(* IEC 61131-3 sources: std_i2980_v2.06_cp053/Source/IMM/ieccontrol/ODC1 (part 5) *)

         IF bAllParallelOpenColumnsReady THEN
            fbDebugTrace2(nODCInterpreter, CONCAT('found fulfilled EndParallelOpen in column ',
                                                 DINT_TO_STRING(i),' -> increase row'));
            bIncreaseRow := TRUE;
         END_IF;

      ELSIF (MoveId  = cMoveNone) AND (MoveDir = cMoveNone) AND (DeviceId.CompId = cCompNone) THEN
         bIncreaseRow := TRUE;
         fbDebugTrace2(nODCInterpreter, CONCAT('at pos:', DINT_TO_STRING(iRow), '/',
                                               DINT_TO_STRING(i), ' empty movement'));

      ELSIF MoveId = cMoveBeginSequence OR MoveId = cMoveEndSequence THEN
         (* skip begin/end sequence markers *)
         bIncreaseRow := TRUE;

      ELSIF MoveId = cMoveStartCondition THEN
         (* start condition *)
         aCheckStartConditionReached(iInstance := sv_ODCSequenceInt[i][iRow].iCount);

         //check safety array of startcondition as long as start condition is not reached
         IF NOT aCheckStartConditionReached.bReached THEN
            abODCCheckDependencies.aCheck.StepPos.iColumn := i;
            abODCCheckDependencies.aCheck.StepPos.iRow := iRow;

            abODCCheckDependencies.aCheck(DeviceIdSelf := DeviceId);
            IF NOT abODCCheckDependencies.aCheck.bAllowed THEN
               fbDebugTrace2(nODCInterpreter, CONCAT('start condition at pos ', DINT_TO_STRING(iRow),
                                                     '/', DINT_TO_STRING(i),
                                                     ' not allowed by safety calculation'));
               aStopInterpreterError();
            END_IF;
         END_IF;

         bIncreaseRow := aCheckStartConditionReached.bReached;

      ELSIF MoveId = cMoveCheckCondition THEN
         (* check condition *)
         aCheckConditionSupervision(iInstance := sv_ODCSequenceInt[i][iRow].iCount);
         bIncreaseRow := aCheckConditionSupervision.bContinue;

      ELSIF (MoveId = cMoveIf) OR (MoveId = cMoveElse) THEN
         (* if or else *)
         aCheckIfCondition(iInstance := sv_ODCSequenceInt[i][iRow].iCount);
         bIncreaseRow := TRUE;
         IF MoveId = cMoveIf THEN
            //programmed "if"
            bGoToEndIf := NOT aCheckIfCondition.bConditionOk;
         ELSE
            //programmed "else"
            bGoToEndIf := aCheckIfCondition.bConditionOk;
         END_IF;
      ELSIF (MoveId = cMoveBeginLoop) THEN
         //check loop condition
         iInstance := sv_ODCSequenceInt[i][iRow].iCount;
         aCheckLoopCondition(iInstance := iInstance);
         IF aCheckLoopCondition.bConditionOk THEN
            //leave the loop
            bGoToEndLoop := TRUE;
            bIncreaseRow := TRUE;
         ELSE
            //increase loop counter and go to next step
            mLoopHelpData[iInstance].iActCount := mLoopHelpData[iInstance].iActCount + 1;
            bGoToEndLoop := FALSE;
            bIncreaseRow := TRUE;
         END_IF;
      ELSIF (MoveId = cMoveEndLoop) THEN
         iInstance := sv_ODCSequenceInt[i][iRow].iCount;
         aCheckLoopCondition(iInstance := iInstance);
         IF NOT aCheckLoopCondition.bConditionOk AND NOT mbStepMode THEN
            //condition not ok -> go back to start of the loop
            //in step mode the loop is only executed once!
            bGoToBeginLoop := TRUE;
         ELSE
            //reset loop counter
            mLoopHelpData[iInstance].iActCount := 0;
            bGoToBeginLoop := FALSE;
         END_IF;

         bIncreaseRow := TRUE;
      ELSE
         // "normal movement"
         (* Flags:
            bIsWaitStep           -> do not start, wait for pos reached
            NOT pbActivated       -> completely skip movement (do not start, do not wait)(checked once when step is activated)
            bContinueWithoutReady -> start, do not wait for ready/pos reached *)

         MoveData := sv_MovementsAvailable[sv_ODCSequenceInt[i][iRow].iMoveNumber].pMovementData;

         //check if device/movement is activated
         IF NOT odcParallelInfo[i].bActivatedChecked THEN
            aCheckActivated(DeviceId := DeviceId,
                            MoveData := MoveData^);

            odcParallelInfo[i].bActivated := aCheckActivated.bActivated;
            odcParallelInfo[i].bActivatedChecked := TRUE;

            IF NOT odcParallelInfo[i].bActivated THEN
               //step not activated -> go to next line
               bIncreaseRow := TRUE;
            END_IF;

            //check if array with PosReached information is available (for instanceabale movements)
            odcParallelInfo[i].bPosReachedArrayLinked := CHECK_REF(MoveData^.InstanceData.pPosReachedArray^);
            odcParallelInfo[i].bMovementReadyArrayLinked := CHECK_REF(MoveData^.InstanceData.pMovementReadyArray^);
         END_IF; //bActivatedChecked

         IF odcParallelInfo[i].bActivated THEN
            (* step is activated *)
            IF odcParallelInfo[i].bSkipAlreadyPosReached THEN
               (* This flag is propagated to new parallel branches
                  and joined (AND) on end of parallel branch
                  Value TRUE:
                  We first check for pos reached
                  - Pos reached: go to the next step
                  - Pos not reached: start movement like we normally do and reset the flag
                    for the current branch
                  Value FALSE:
                  We act normally and start the movement *)

               IF odcParallelInfo[i].bPosReachedArrayLinked THEN
                  iInstance := sv_ODCSequenceInt[i][iRow].iCount;
                  IF MoveData^.InstanceData.pPosReachedArray^[iInstance] THEN
                     bIncreaseRow := TRUE;
                  END_IF;
               ELSE
                  fbCheckPosReached(DeviceId := DeviceId,
                                 MoveDir  := MoveDir,
                                 MoveId   := MoveId);
                  IF fbCheckPosReached.bPosReached THEN
                     bIncreaseRow := TRUE;
                  END_IF;
               END_IF;

               IF bIncreaseRow THEN
                  fbDebugTrace2(nODCInterpreter, CONCAT('at pos:', DINT_TO_STRING(iRow), '/',
                                          DINT_TO_STRING(i), ' skipping movement ',
                                          DINT_TO_STRING(DeviceId.CompId), '.',
                                          DINT_TO_STRING(DeviceId.IndexId), ' ',
                                          DINT_TO_STRING(MoveId), '/',
                                          DINT_TO_STRING(MoveDir), ' pos:',
                                          DINT_TO_STRING(sv_ODCSequenceInt[i][iRow].iCount),
                                          ' because it already has PosReached TRUE'));
               ELSE
                  (* pos not reached -> start the movement
                  and continue normal execution from here *)
                  fbDebugTrace2(nODCInterpreter, CONCAT('at pos:', DINT_TO_STRING(iRow), '/',
                                    DINT_TO_STRING(i), ' disable skipping PosReached movements ',
                                    DINT_TO_STRING(DeviceId.CompId), '.',
                                    DINT_TO_STRING(DeviceId.IndexId), ' ',
                                    DINT_TO_STRING(MoveId), '/',
                                    DINT_TO_STRING(MoveDir), ' pos:',
                                    DINT_TO_STRING(sv_ODCSequenceInt[i][iRow].iCount),
                                    ' because it has PosReached FALSE'));
                  odcParallelInfo[i].bSkipAlreadyPosReached := FALSE;
               END_IF;

            END_IF;

            (* start the movement *)
            IF odcParallelInfo[i].bSkipAlreadyPosReached THEN
               (* bSkipAlreadyPosReached is still set -> the current movement already has PosReached TRUE *)
               (* -> we do not need to start it *)
               ;
            ELSIF MoveData^.bIsWaitStep THEN
               (* do not start movement, just wait for pos reached *)
               odcParallelInfo[i].bStartSent := TRUE;

            ELSIF NOT odcParallelInfo[i].bStartSent THEN
               bConditionLinked := CHECK_REF(MoveData^.pbStartConditionReached^);
               IF (bConditionLinked AND MoveData^.pbStartConditionReached^) OR NOT bConditionLinked THEN
                  // pbStartConditionReached reached or not linked -> start movement

                  fbDebugTrace2(nODCInterpreter, CONCAT('at pos:', DINT_TO_STRING(iRow), '/',
                                                         DINT_TO_STRING(i), ' checking dependencies for movement ',
                                                         DINT_TO_STRING(DeviceId.CompId), '.',
                                                         DINT_TO_STRING(DeviceId.IndexId), ' ',
                                                         DINT_TO_STRING(MoveId), '/',
                                                         DINT_TO_STRING(MoveDir)));

                  abODCCheckDependencies.aCheck.StepPos.iColumn := i;
                  abODCCheckDependencies.aCheck.StepPos.iRow := iRow;

                  abODCCheckDependencies.aCheck(DeviceIdSelf := DeviceId);
                  IF NOT abODCCheckDependencies.aCheck.bAllowed THEN
                     (* evCheckLocklist makes sure other alarms(caused by FBLockUnlock for this movement are also set *)
                     evCheckLocklistEventData.DeviceId := DeviceId;
                     evCheckLocklistEventData.MoveId   := MoveId;
                     evCheckLocklistEventData.MoveDir  := MoveDir;
                     fbDebugTrace2(nODCInterpreter, CONCAT('movement ', DINT_TO_STRING(MoveId),
                                                           '/', DINT_TO_STRING(MoveDir),
                                                           ' not allowed by safety calculation -> sending evCheckLocklist to view all other alarms'));
                     SET_EVENT(evCheckLocklist, evCheckLocklistEventData);
                     aStopInterpreterError();
                  ELSE // NOT abODCCheckDependencies.aCheck.bAllowed
                     (* dependencies OK *)
                     fbDebugTrace2(nODCInterpreter, CONCAT('at pos:', DINT_TO_STRING(iRow), '/',
                                                            DINT_TO_STRING(i), ' starting movement ',
                                                            DINT_TO_STRING(DeviceId.CompId), '.',
                                                            DINT_TO_STRING(DeviceId.IndexId), ' ',
                                                            DINT_TO_STRING(MoveId), '/',
                                                            DINT_TO_STRING(MoveDir), ' ',
                                                            DINT_TO_STRING(sv_ODCSequenceInt[i][iRow].iCount)));

                     aAddStartedManualMovement.StepPos.iColumn := i;
                     aAddStartedManualMovement.StepPos.iRow := iRow;
                     aAddStartedManualMovement(DeviceId := DeviceId,
                                                MoveId   := MoveId,
                                                MoveDir  := MoveDir,
                                                iInstance := sv_ODCSequenceInt[i][iRow].iCount);

                        (* try to start the movement *)
                     IF aAddStartedManualMovement.bOK THEN
                        odcParallelInfo[i].bStartSent := TRUE;

                        //save time when start event was sent
                        odcParallelInfo[i].dStartTime := fbRTC.CDT;

                        fbStart(DeviceId := DeviceId,
                                 MoveDir  := MoveDir,
                                 MoveId   := MoveId,
                                 IntermediateCond := sv_ODCSequenceInt[i][iRow].iCount);
                     ELSE
                        aStopInterpreterError();
                     END_IF;
                  END_IF; // NOT fbODCCheckDependencies.bAllowed

               ELSE // (bConditionLinked AND MoveData^.pbStartConditionReached^) OR NOT bConditionLinked
                  IF NOT odcParallelInfo[i].bStartConditionWarnPrinted THEN
                     IF sv_TraceLevel.bODCInterpreter THEN
                        dummy := Print('at pos:%d/%d waiting for pbStartConditionReached before starting movement %d.%d %d/%d',
                                    iRow, i, DeviceId.CompId, DeviceId.IndexId, MoveId, MoveDir);
                     END_IF;
                     odcParallelInfo[i].bStartConditionWarnPrinted := TRUE;
                  END_IF;
               END_IF; // pbStartConditionReached^
            END_IF; // NOT odcParallelInfo[i].bStartSent

            (* now wait for the movement to finish *)
            IF odcParallelInfo[i].bSkipAlreadyPosReached THEN
               ;
            ELSIF MoveData^.bIsWaitStep THEN
               (* movement was never started, only wait for pos reached, not for ready
                  otherwise we have a problem when we wait for a certain pos reached
                  but we are still moving to another position
                  (example: mold close, wait for intermediate pos) *)
               IF odcParallelInfo[i].bPosReachedArrayLinked THEN
                  iInstance := sv_ODCSequenceInt[i][iRow].iCount;
                  bIncreaseRow := MoveData^.InstanceData.pPosReachedArray^[iInstance];
               ELSE
                  fbCheckPosReached(DeviceId := DeviceId,
                                    MoveDir  := MoveDir,
                                    MoveId   := MoveId);
                  IF fbCheckPosReached.bPosReached THEN
                     bIncreaseRow := TRUE;
                  END_IF;
               END_IF;

            ELSIF odcParallelInfo[i].bStartSent THEN
               (* start event was sent -> we can now wait for the movement to finish *)
               IF MoveData^.bContinueWithoutReady THEN
                  (* do not wait for the movement to finish, continue immediately
                     useful for air valves *)
                  bIncreaseRow := TRUE;
               ELSE
                  (* normal movement
                     check if the movement is finished(ready),
                     and if pos is reached(when the movement has a pos reached variable) *)
                  IF MoveData^.bInstanceable AND odcParallelInfo[i].bMovementReadyArrayLinked THEN
                     iInstance := sv_ODCSequenceInt[i][iRow].iCount;
                     bMovementReady := MoveData^.InstanceData.pMovementReadyArray^[iInstance];
                  ELSE
                     fbCheckReady(DeviceId := DeviceId);
                     bMovementReady := fbCheckReady.bReady;
                  END_IF;

                  IF bMovementReady THEN
                     aCheckPosReached(DeviceId := DeviceId,
                                      MoveId := MoveId,
                                      MoveDir := MoveDir,
                                      iColumn := i,
                                      iRow := iRow);

                     IF aCheckPosReached.bPosReachedOk THEN
                        // everything ok -> correct duration and go to next row
                        aCorrectDuration(pMoveData := MoveData,
                                         iColumn := i,
                                         DeviceId := DeviceId);

                        bIncreaseRow := TRUE;
                     END_IF;

                  END_IF; // check ready
               END_IF; // MoveData^.bContinueWithoutReady
            END_IF; // start condition reached
         END_IF; // step activated
      END_IF; //movement ID

      IF bIncreaseRow THEN
         // set step state to Ready
         IF sv_ODCSequenceInt[i][odcParallelInfo[i].iRow].StepState <> nStateError THEN
            // do not reset steps with error flag
            IF NOT CHECK_REF(MoveData^) OR NOT MoveData^.bContinueWithoutReady THEN
               fbSetStepState.StepPos.iRow := odcParallelInfo[i].iRow;
               fbSetStepState.StepPos.iColumn := i;
               fbSetStepState(StepState := nStateReady);
            END_IF;
         END_IF;

         IF bGoToEndIf THEN
            aGoToEndIf(iColumn := i);
         ELSIF bGoToBeginLoop THEN
            bGoToBeginLoop := FALSE;
            aGoToBeginLoop(iColumn := i, iInstance := sv_ODCSequenceInt[i][iRow].iCount);
         ELSIF bGoToEndLoop THEN
            bGoToEndLoop := FALSE;
            aGoToEndLoop(iColumn := i, iInstance := sv_ODCSequenceInt[i][iRow].iCount);
         ELSE
            aIncreaseRow(iColumn := i, iEndRow := miEndRow);
         END_IF;
      END_IF;
   END_IF; //odcParallelInfo[i].bColumnActive
END_FOR;

//interesting for HMI to see state of the interpreter
sv_InterpreterParallelInfo := odcParallelInfo;

;#END_EDIT_BLOCK END_ALGORITHM

(*
Search a Movement in the ODC array by DeviceId, MoveId and MovedDir
and return the position in the array.

If bAllowNonMatchingId is TRUE only DeviceId and MoveDir need to match.
But it still tries to get the best match(MoveId equals)

If IntermediateCond is <> 0, it is also checked against iCount when checking for exact match.

When a movement is found bFound is TRUE and StepPos contains the position
of the movement in the ODC array
*)

ALGORITHM aFindLabel

VAR_INPUT
 DeviceId : tsDeviceId (* DeviceId of the movement to search for *);
 MoveId : tMoveIdent (* MoveId of the movement to search for *);
 MoveDir : tMoveIdent (* MoveDir of the movement to search for *);
 IntermediateCond : DINT (* Intermediate condition to search for *);
 bAllowNonMatchingId : BOOL (* Also return a match if MoveId is different *);
 SearchStartPos : tsODCStepPos (* startposition for searching *);
END_VAR

VAR_OUTPUT
 StepPos : tsODCStepPos (* Position in ODC array wher the movement was found *);
 bFound : BOOL (* TRUE if a movement was found *);
END_VAR

VAR_TEMP
 iTmpRow : DINT;
 iTmpColumn : DINT;
 iSearchColumn : DINT;
END_VAR
#BEGIN_EDIT_BLOCK
(**************************************** WARNING ********************************************
 *** The KEBA Kemro K2 System including software is not intended for safety control tasks! ***
 ***                       For further information see Comment tab!                        ***
 *********************************************************************************************)

bFound := FALSE;
StepPos.iColumn := 0;
StepPos.iRow := 0;

FOR iTmpRow := SearchStartPos.iRow TO sv_iUsedRows DO

   IF iTmpRow = SearchStartPos.iRow THEN
      //start searching in the given column
      iSearchColumn := SearchStartPos.iColumn;
   ELSE
      //start searching in the first column
      iSearchColumn := 1;
   END_IF;

   FOR iTmpColumn := iSearchColumn TO sv_iUsedColumns DO
      IF sv_ODCSequence[iTmpColumn][iTmpRow].iCompId = DeviceId.CompId AND
         INT_TO_DINT(sv_ODCSequence[iTmpColumn][iTmpRow].iIndexId) = DeviceId.IndexId THEN
         IF sv_ODCSequence[iTmpColumn][iTmpRow].iMoveId = MoveId AND
            sv_ODCSequence[iTmpColumn][iTmpRow].iMoveDir = MoveDir AND
            (IntermediateCond = 0 OR // do not care about intermediate condion if we don't search for it?
                                     // FIXME check flag in MoveData instead??
             INT_TO_DINT(sv_ODCSequence[iTmpColumn][iTmpRow].iCount) = IntermediateCond) THEN
            fbDebugTrace2(nODCInterpreter, CONCAT('found exact match of MoveId ',
                                                  DINT_TO_STRING(DeviceId.CompId),
                                                  '.',
                                                  DINT_TO_STRING(DeviceId.IndexId),
                                                  ' ',
                                                  DINT_TO_STRING(MoveId),
                                                  '/',
                                                  DINT_TO_STRING(MoveDir),
                                                  ' ',
                                                  DINT_TO_STRING(IntermediateCond),
                                                  ' at pos:',
                                                  DINT_TO_STRING(iTmpRow),
                                                  '/',
                                                  DINT_TO_STRING(iTmpColumn)));

            StepPos.iColumn := iTmpColumn;
            StepPos.iRow := iTmpRow;
            bFound := TRUE;
            RETURN;

         ELSIF bAllowNonMatchingId AND sv_ODCSequence[iTmpColumn][iTmpRow].iMoveDir = MoveDir THEN
            fbDebugTrace2(nODCInterpreter, CONCAT('found NON exact match of MoveId ',
                                                  DINT_TO_STRING(DeviceId.CompId),
                                                  '.',
                                                  DINT_TO_STRING(DeviceId.IndexId),
                                                  ' ',
                                                  DINT_TO_STRING(MoveId),
                                                  '/',
                                                  DINT_TO_STRING(MoveDir),
                                                  ' ',
                                                  DINT_TO_STRING(IntermediateCond),
                                                  ' at pos:',
                                                  DINT_TO_STRING(iTmpRow),
                                                  '/',
                                                  DINT_TO_STRING(iTmpColumn)));
            StepPos.iColumn := iTmpColumn;
            StepPos.iRow := iTmpRow;
            bFound := TRUE;
         END_IF;
      END_IF;
   END_FOR;
END_FOR;

IF NOT bFound THEN
   fbDebugTrace2(nODCInterpreter, CONCAT('movement ',
                                          DINT_TO_STRING(DeviceId.CompId),
                                          '.',
                                          DINT_TO_STRING(DeviceId.IndexId),
                                          ' ',
                                          DINT_TO_STRING(MoveId),
                                          '/',
                                          DINT_TO_STRING(MoveDir),
                                          ' ',
                                          DINT_TO_STRING(IntermediateCond),
                                          ' not found in auto cycle'));
END_IF;

;#END_EDIT_BLOCK END_ALGORITHM

(*
Notify the Interpreter that the array has been reinitialized
(this clears the fatal error flag)
*)

ALGORITHM aSetInitOK

VAR
 DeviceIdAll : tsDeviceId;
END_VAR
#BEGIN_EDIT_BLOCK
(**************************************** WARNING ********************************************
 *** The KEBA Kemro K2 System including software is not intended for safety control tasks! ***
 ***                       For further information see Comment tab!                        ***
 *********************************************************************************************)

IF mbFatalError THEN
   mbFatalError := FALSE;

   (* unlock all movements locked by aStopInterpreterInternal *)
   DeviceIdAll.CompId := cCompAll;
   DeviceIdAll.IndexId := cAllDevIndex;

   fbLockUnlock(DeviceId := DeviceIdAll,
               MoveDir  := cMoveAll,
               MoveId   := cMoveAll,
               Mode     := nUnlock);
END_IF;

;#END_EDIT_BLOCK END_ALGORITHM

(*
Actual status of the interpreter.
*)

ALGORITHM aStatus

VAR_OUTPUT
 bActive : BOOL (* Interpreter is currently executing a ODC array *);
 bError : BOOL (* Interpreter is stopped, because a error happened during interpreting *);
 bFinished : BOOL (* Interpreter is stopped, because it reached the end of the array *);
END_VAR
#BEGIN_EDIT_BLOCK
(**************************************** WARNING ********************************************
 *** The KEBA Kemro K2 System including software is not intended for safety control tasks! ***
 ***                       For further information see Comment tab!                        ***
 *********************************************************************************************)

bError := mbFatalError OR mbNormalError;
bFinished := mbFinished;
bActive := mbActive;

;#END_EDIT_BLOCK END_ALGORITHM

ALGORITHM aInterruptSequence

VAR_TEMP
 i : DINT;
END_VAR

VAR
 StartedMovements : tsStartedMoveDataODCExtended;
 fbStop : FBStop;
 iMoveNr : DINT;
 fbGetMoveNumber : FBGetMoveNumber;
END_VAR
#BEGIN_EDIT_BLOCK
(**************************************** WARNING ********************************************
 *** The KEBA Kemro K2 System including software is not intended for safety control tasks! ***
 ***                       For further information see Comment tab!                        ***
 *********************************************************************************************)

mbStepMode := TRUE;

//stop started movements
StartedMovements := sv_StartedManualMovements;
FOR i := 1 TO StartedMovements.iStartedMovements DO

   //get move number
   fbGetMoveNumber(DeviceId := StartedMovements.MoveData[i].DeviceId,
                   MoveId := StartedMovements.MoveData[i].MoveId,
                   MoveDir := StartedMovements.MoveData[i].MoveDir,
                   iMoveNumber => iMoveNr);

   IF NOT sv_MovementsAvailable[iMoveNr].pMovementData^.bFinishAtInterrupt THEN
      //stop movement
      fbStop(DeviceId := StartedMovements.MoveData[i].DeviceId);
   ELSE
      //movement should finish
      //increase number of active row because otherwise this movement is started
      //again when stepping fwd
      aIncreaseRow(iColumn := StartedMovements.MoveData[i].StepPos.iColumn,
                   iEndRow := miEndRow);
   END_IF;

END_FOR;

//disable steps
FOR i := 1 TO cMaxParallelMovements DO
   IF odcParallelInfo[i].bColumnActive THEN
      odcParallelInfo[i].bDisabled := TRUE;
   END_IF;
END_FOR;

mbActive := FALSE;

sv_InterpreterParallelInfo := odcParallelInfo;

;#END_EDIT_BLOCK END_ALGORITHM

ALGORITHM aContinueSequence

VAR_TEMP
 i : DINT;
END_VAR

VAR
 fbSetStepState : FBSetStepState;
END_VAR
#BEGIN_EDIT_BLOCK
(**************************************** WARNING ********************************************
 *** The KEBA Kemro K2 System including software is not intended for safety control tasks! ***
 ***                       For further information see Comment tab!                        ***
 *********************************************************************************************)

//reset relevant flags
FOR i := 1 TO cMaxParallelMovements DO
   IF odcParallelInfo[i].bColumnActive THEN
      odcParallelInfo[i].bStartSent := FALSE;
      odcParallelInfo[i].bStartConditionWarnPrinted := FALSE;
      odcParallelInfo[i].bActivatedChecked := FALSE;
      odcParallelInfo[i].bDisabled := FALSE;

      //set step state to "active"
      fbSetStepState.StepPos.iColumn := i;
      fbSetStepState.StepPos.iRow := odcParallelInfo[i].iRow;
      fbSetStepState(StepState := nStateActive);
   END_IF;

END_FOR;

mbActive := TRUE;
mbStepMode := FALSE;

;#END_EDIT_BLOCK END_ALGORITHM

ALGORITHM aEnableNextStep

VAR_TEMP
 i : DINT;
END_VAR
#BEGIN_EDIT_BLOCK
(**************************************** WARNING ********************************************
 *** The KEBA Kemro K2 System including software is not intended for safety control tasks! ***
 ***                       For further information see Comment tab!                        ***
 *********************************************************************************************)

//enable steps
FOR i := 1 TO cMaxParallelMovements DO
   IF odcParallelInfo[i].bColumnActive THEN
      odcParallelInfo[i].bDisabled := FALSE;
      odcParallelInfo[i].bStartSent := FALSE;
      odcParallelInfo[i].bStartConditionWarnPrinted := FALSE;
      odcParallelInfo[i].bActivatedChecked := FALSE;

      //set step state to "active"
      fbSetStepState.StepPos.iColumn := i;
      fbSetStepState.StepPos.iRow := odcParallelInfo[i].iRow;
      fbSetStepState(StepState := nStateActive);
   END_IF;

END_FOR;

mbActive := TRUE;

;#END_EDIT_BLOCK END_ALGORITHM

ALGORITHM aResetStepMode

#BEGIN_EDIT_BLOCK
(**************************************** WARNING ********************************************
 *** The KEBA Kemro K2 System including software is not intended for safety control tasks! ***
 ***                       For further information see Comment tab!                        ***
 *********************************************************************************************)

mbStepMode := FALSE;

;#END_EDIT_BLOCK END_ALGORITHM

ALGORITHM aDecreaseRow

VAR_INPUT
 bStartInActualLine : BOOL (* TRUE: start in actual line; FALSE: start in (actual line - 1) *);
 iColumn : DINT;
 iEndRow : DINT;
END_VAR

VAR_OUTPUT
 iNewActivatedColumn : DINT;
END_VAR

VAR_TEMP
 iTmpLine : DINT;
 iTmpColumn : DINT;
 x : DINT;
 iLine : DINT;
END_VAR

VAR
 iMoveId : tMoveIdent;
 fbSetStepState : FBSetStepState;
 bParallelTreeReady : BOOL;
 bOk : BOOL;
 bContinueDecreasing : BOOL;
 iStartRow : DINT;
 iCount : INT;
END_VAR
#BEGIN_EDIT_BLOCK
(**************************************** WARNING ********************************************
 *** The KEBA Kemro K2 System including software is not intended for safety control tasks! ***
 ***                       For further information see Comment tab!                        ***
 *********************************************************************************************)

IF bStartInActualLine THEN
   iStartRow := odcParallelInfo[iColumn].iRow;
ELSE
   iStartRow := (odcParallelInfo[iColumn].iRow - 1);
END_IF;

//reset step state of actually active step
fbSetStepState.StepPos.iColumn := iColumn;
fbSetStepState.StepPos.iRow := odcParallelInfo[iColumn].iRow;
fbSetStepState(StepState := nStateDefault);

iNewActivatedColumn := 0;

//get next line with a "real" movement
FOR iTmpLine := iStartRow TO iEndRow BY -1 DO
   fbDebugTrace2(nODCInterpreter, CONCAT('decreasing IP of column ', DINT_TO_STRING(iColumn),
                                         ' to ', DINT_TO_STRING(iTmpLine)));

   iMoveId := sv_ODCSequence[iColumn][iTmpLine].iMoveId;

   IF (iMoveId = cMoveEndIf) THEN
      // end_if => check if this "if" instance is active or already completely executed
      iCount := sv_ODCSequence[iColumn][iTmpLine].iCount;
      IF (mIFConditionHelpData[iCount].iInternalCount < 2) THEN
         //if or else tree is active
         //set active line in this column to begin of this "if" or "else"
         //so that stepping bwd can continue before this "if / else"
         FOR iLine := (iTmpLine - 1) TO 1 BY -1 DO
            IF ((sv_ODCSequence[iColumn][iLine].iMoveId = cMoveIf) OR (sv_ODCSequence[iColumn][iLine].iMoveId = cMoveElse)) AND
               (sv_ODCSequence[iColumn][iLine].iCount = iCount) THEN
               odcParallelInfo[iColumn].iRow := (iLine - 1);  //set row to "start parallel" step
               EXIT;
            END_IF;
         END_FOR;
         mIFConditionHelpData[iCount].iInternalCount := (mIFConditionHelpData[iCount].iInternalCount - 1);
      ELSE
         //condition completely executed -> do not allow stepping into
         odcParallelInfo[iColumn].iRow := (iTmpLine + 1); //set row to "end parallel" step
         odcParallelInfo[iColumn].bDisabled := TRUE;
         SET_ALARM(Name := erNoStepBwdIntoCondition);
      END_IF;

      EXIT;
   ELSIF (iMoveId = cMoveEndLoop) THEN
      // end loop => stop stepping bwd here
      odcParallelInfo[iColumn].iRow := iTmpLine; //set row to "end loop" step
      odcParallelInfo[iColumn].bDisabled := TRUE;
      SET_ALARM(Name := erNoStepBwdIntoLoop);
      EXIT;
   ELSIF (iMoveId = cMoveBeginLoop) THEN
      // begin of loop => stop stepping bwd here (do not modify line number)
      odcParallelInfo[iColumn].bDisabled := TRUE;
      SET_ALARM(Name := erNoStepBwdOutOfLoop);
      EXIT;
   ELSIF (iMoveId = cMoveBeginSequence) OR (iMoveId = cMoveEndSequence) THEN
      ; // begin or end sequence
   ELSIF (iMoveId = cMoveNone) OR (iMoveId = cMoveBeginGroup) OR (iMoveId = cMoveEndGroup) THEN
      ; //empty step or begin group / end group
   ELSIF (iMoveId = cMoveIf) OR (iMoveId = cMoveElse) THEN
      ; //if , else
   ELSIF iMoveId = cMoveEndParallelOpen THEN
      ; //no special action necessary
   ELSIF iMoveId = cMoveEndParallel THEN
      //get according column and activate it
      FOR iTmpColumn := (iColumn + 1) TO sv_iUsedColumns DO
         IF sv_ODCSequence[iTmpColumn][iTmpLine].iMoveId = cMoveEndParallel THEN
            odcParallelInfo[iTmpColumn].bColumnActive := TRUE;
            odcParallelInfo[iTmpColumn].iRow := (iTmpLine + 1); //necessary to handle more end parallel in one line
            odcParallelInfo[iTmpColumn].bDisabled := TRUE;
            iNewActivatedColumn := iTmpColumn;
            EXIT;
         END_IF;
      END_FOR;
   ELSIF (iMoveId = cMoveStartParallel) OR (iMoveId = cMoveStartParallelOpen) THEN
      bContinueDecreasing := FALSE;
      FOR iTmpColumn := 1 TO sv_iUsedColumns DO
         IF (sv_ODCSequence[iTmpColumn][iTmpLine].iMoveId = cMoveStartParallel) OR
            (sv_ODCSequence[iTmpColumn][iTmpLine].iMoveId = cMoveStartParallelOpen) THEN

            //start parallel or start parallel open found
            IF iTmpColumn < iColumn THEN
               //SP left to actual column found
               //-> deactivate actual column and set line number
               odcParallelInfo[iColumn].iRow := iTmpLine;
               odcParallelInfo[iColumn].bDisabled := FALSE;
               odcParallelInfo[iColumn].bColumnActive := FALSE;
               IF sv_TraceLevel.bODCInterpreter THEN
                  dummy := Print('aDecreaseRow: deactivate column %d ',iColumn);
               END_IF;
            ELSE
               //SP is the most left one in this line
               //-> all SP to the right must be deactivated and their active row must be equal
               bOk := TRUE;
               FOR x := (iTmpColumn + 1) TO sv_iUsedColumns DO
                  //only consider SP entries
                  IF (sv_ODCSequence[x][iTmpLine].iMoveId = cMoveStartParallel) OR
                     (sv_ODCSequence[x][iTmpLine].iMoveId = cMoveStartParallelOpen) THEN
                     bParallelTreeReady := NOT odcParallelInfo[x].bColumnActive AND (odcParallelInfo[x].iRow = iTmpLine);
                     bOk := bOk AND bParallelTreeReady;
                  END_IF;
               END_FOR;

               IF bOk THEN
                  //all parallel trees ready -> decrease line of this column so that it can continue
                  bContinueDecreasing := TRUE;
               ELSE
                  //column still active -> wait in this line
                  odcParallelInfo[iColumn].iRow := iTmpLine;
                  odcParallelInfo[iColumn].bDisabled := TRUE;
                  bContinueDecreasing := FALSE;
               END_IF;
            END_IF;

            EXIT; //exit inner loop
         END_IF;
      END_FOR;

      IF NOT bContinueDecreasing THEN
         EXIT;  // exit outer loop
      END_IF;
   ELSE
      //valid step found -> set line number and disable this step
      IF sv_TraceLevel.bODCInterpreter THEN
         dummy := Print('///////// set active row of column %d to %d ////////////',iColumn, iTmpLine);
      END_IF;
      odcParallelInfo[iColumn].iRow := iTmpLine;
      odcParallelInfo[iColumn].bDisabled := TRUE;
      EXIT;
   END_IF;
END_FOR;

odcParallelInfo[iColumn].bStartSent := FALSE;
odcParallelInfo[iColumn].bStartConditionWarnPrinted := FALSE;
odcParallelInfo[iColumn].bActivatedChecked := FALSE;
odcParallelInfo[iColumn].bPosReachedArrayLinked := FALSE;
odcParallelInfo[iColumn].bMovementReadyArrayLinked := FALSE;

sv_InterpreterParallelInfo[iColumn] := odcParallelInfo[iColumn];

;#END_EDIT_BLOCK END_ALGORITHM

END_ALGORITHM_BLOCK

#END_OF_IEC_PART

@Puma @IecEditor 6 96 @Pou 25
@@@BEG_Comment@@@
@h    ! WARNING !
@h    The Kemro K2 system (including software) only meets category B according to EN 954-1,
@h    thus it is not intended for usage in safety-relevant control applications in the field
@h    of personal safety (e.g. emergency stop).
@h    To implement potentially necessary safety-relevant control tasks, always use additional
@h    external safety devices that are intended for the particular purpose, and meet the necessary
@h    functional safety.
@h    For further information see EN 954-1 (EN ISO 13849-1) and/or the K2-x00 user manual, chapter
@h    "CE conformity, directives and standards".
@@@END_Comment@@@

@BEG_Contents

@BEG_Func
@RT(17)FuncTreeContainer
4
@Var @RT(9)CHECK_REF @RT(0) @T @T @DERIVED 0 @F @RT(23)KEBA_STANDARD_PROCEDURE @F
@T
@BEG_Attrib
0 @RT(0) @RT(0)
@END_Attrib
1 1 @F @F @F @F

@Var @RT(9)SET_EVENT @RT(0) @T @T @DERIVED 0 @F @RT(23)KEBA_STANDARD_PROCEDURE @F
@T
@BEG_Attrib
0 @RT(0) @RT(0)
@END_Attrib
1 1 @F @F @F @F

@Var @RT(9)SET_ALARM @RT(0) @T @T @DERIVED 0 @F @RT(23)KEBA_STANDARD_PROCEDURE @F
@T
@BEG_Attrib
0 @RT(0) @RT(0)
@END_Attrib
1 1 @F @F @F @F

@Var @RT(11)RESET_ALARM @RT(0) @T @T @DERIVED 0 @F @RT(23)KEBA_STANDARD_PROCEDURE @F
@T
@BEG_Attrib
0 @RT(0) @RT(0)
@END_Attrib
1 1 @F @F @F @F

@END_Func

@BEG_Const
@RT(18)ConstTreeContainer
25
@Var @RT(21)cMaxParallelMovements @RT(0) @T @F @DT @RT(4)DINT @RT(0) @T @T @BASIC 0 @F
@F @F
@T
@BEG_Attrib
0 @RT(1)6 @RT(62)maximum number of columns in odc array (<=cMaxActiveMovements)
@END_Attrib
1 1 @F @F @F @F

@Var @RT(12)cMaxODCSteps @RT(0) @T @F @DT @RT(4)DINT @RT(0) @T @T @BASIC 0 @F
@F @F
@T
@BEG_Attrib
0 @RT(3)100 @RT(35)maximum number of rows in odc array
@END_Attrib
1 1 @F @F @F @F

@Var @RT(9)cMoveNone @RT(0) @T @F @DT @RT(4)DINT @RT(0) @T @T @BASIC 0 @F
@F @F
@T
@BEG_Attrib
0 @RT(13)cMinMoveIdent @RT(4)None
@END_Attrib
1 1 @F @F @F @F

@Var @RT(18)cMoveStartParallel @RT(0) @T @F @DT @RT(4)DINT @RT(0) @T @T @BASIC 0 @F
@F @F
@T
@BEG_Attrib
0 @RT(2)45 @RT(34)dummy movement for "StartParallel"
@END_Attrib
1 1 @F @F @F @F

@Var @RT(12)cCompEjector @RT(0) @T @F @DT @RT(4)DINT @RT(0) @T @T @BASIC 0 @F
@F @F
@T
@BEG_Attrib
0 @RT(3)102 @RT(17)Component Ejector
@END_Attrib
1 1 @F @F @F @F

@Var @RT(24)cCompCentralCoordination @RT(0) @T @F @DT @RT(4)DINT @RT(0) @T @T @BASIC 0 @F
@F @F
@T
@BEG_Attrib
0 @RT(3)106 @RT(29)Component CentralCoordination
@END_Attrib
1 1 @F @F @F @F

@Var @RT(13)cCompAirValve @RT(0) @T @F @DT @RT(4)DINT @RT(0) @T @T @BASIC 0 @F
@F @F
@T
@BEG_Attrib
0 @RT(3)118 @RT(19)Component Air Valve
@END_Attrib
1 1 @F @F @F @F

@Var @RT(8)cMoveFwd @RT(0) @T @F @DT @RT(4)DINT @RT(0) @T @T @BASIC 0 @F
@F @F
@T
@BEG_Attrib
0 @RT(2)12 @RT(16)movement forward
@END_Attrib
1 1 @F @F @F @F

@Var @RT(10)cMoveStart @RT(0) @T @F @DT @RT(4)DINT @RT(0) @T @T @BASIC 0 @F
@F @F
@T
@BEG_Attrib
0 @RT(2)19 @RT(19)start (eg Airvalve)
@END_Attrib
1 1 @F @F @F @F

@Var @RT(8)cMoveBwd @RT(0) @T @F @DT @RT(4)DINT @RT(0) @T @T @BASIC 0 @F
@F @F
@T
@BEG_Attrib
0 @RT(2)11 @RT(17)movement backward
@END_Attrib
1 1 @F @F @F @F

@Var @RT(10)cMoveShake @RT(0) @T @F @DT @RT(4)DINT @RT(0) @T @T @BASIC 0 @F
@F @F
@T
@BEG_Attrib
0 @RT(2)18 @RT(51)shaking movement (for example ejector vibrate mode)
@END_Attrib
1 1 @F @F @F @F

@Var @RT(16)cMoveEndParallel @RT(0) @T @F @DT @RT(4)DINT @RT(0) @T @T @BASIC 0 @F
@F @F
@T
@BEG_Attrib
0 @RT(2)46 @RT(32)dummy movement for "EndParallel"
@END_Attrib
1 1 @F @F @F @F

@Var @RT(16)cMoveEndSequence @RT(0) @T @F @DT @RT(4)DINT @RT(0) @T @T @BASIC 0 @F
@F @F
@T
@BEG_Attrib
0 @RT(2)44 @RT(36)dummy movement for end of a sequence
@END_Attrib
1 1 @F @F @F @F

@Var @RT(8)cCompODC @RT(0) @T @F @DT @RT(4)DINT @RT(0) @T @T @BASIC 0 @F
@F @F
@T
@BEG_Attrib
0 @RT(3)136 @RT(13)Component ODC
@END_Attrib
1 1 @F @F @F @F

@Var @RT(9)cCompNone @RT(0) @T @F @DT @RT(4)DINT @RT(0) @T @T @BASIC 0 @F
@F @F
@T
@BEG_Attrib
0 @RT(10)cMinCompId @RT(4)None
@END_Attrib
1 1 @F @F @F @F

@Var @RT(10)cMinCompId @RT(0) @T @F @DT @RT(4)DINT @RT(0) @T @T @BASIC 0 @F
@F @F
@T
@BEG_Attrib
0 @RT(3)100 @RT(21)minimum Component ID
@END_Attrib
1 1 @F @F @F @F

@Var @RT(10)cMaxCompId @RT(0) @T @F @DT @RT(4)DINT @RT(0) @T @T @BASIC 0 @F
@F @F
@T
@BEG_Attrib
0 @RT(3)250 @RT(21)maximum Component ID
@END_Attrib
1 1 @F @F @F @F

@Var @RT(15)cMaxDeviceIndex @RT(0) @T @F @DT @RT(4)DINT @RT(0) @T @T @BASIC 0 @F
@F @F
@T
@BEG_Attrib
0 @RT(2)10 @RT(39)maximum number of devices per component
@END_Attrib
1 1 @F @F @F @F

@Var @RT(13)cMinMoveIdent @RT(0) @T @F @DT @RT(4)DINT @RT(0) @T @T @BASIC 0 @F
@F @F
@T
@BEG_Attrib
0 @RT(1)1 @RT(32)lower limit for MoveId / MoveDir
@END_Attrib
1 1 @F @F @F @F

@Var @RT(13)cMaxMoveIdent @RT(0) @T @F @DT @RT(4)DINT @RT(0) @T @T @BASIC 0 @F
@F @F
@T
@BEG_Attrib
0 @RT(3)600 @RT(32)upper limit for MoveId / MoveDir
@END_Attrib
1 1 @F @F @F @F

@Var @RT(7)cMoveIf @RT(0) @T @F @DT @RT(4)DINT @RT(0) @T @T @BASIC 0 @F
@F @F
@T
@BEG_Attrib
0 @RT(1)2 @RT(2)IF
@END_Attrib
1 1 @F @F @F @F

@Var @RT(9)cMoveElse @RT(0) @T @F @DT @RT(4)DINT @RT(0) @T @T @BASIC 0 @F
@F @F
@T
@BEG_Attrib
0 @RT(1)3 @RT(4)ELSE
@END_Attrib
1 1 @F @F @F @F

@Var @RT(22)cMoveStartParallelOpen @RT(0) @T @F @DT @RT(4)DINT @RT(0) @T @T @BASIC 0 @F
@F @F
@T
@BEG_Attrib
0 @RT(1)9 @RT(17)StartParallelOpen
@END_Attrib
1 1 @F @F @F @F

@Var @RT(20)cMoveEndParallelOpen @RT(0) @T @F @DT @RT(4)DINT @RT(0) @T @T @BASIC 0 @F
@F @F
@T
@BEG_Attrib
0 @RT(2)10 @RT(15)EndParallelOpen
@END_Attrib
1 1 @F @F @F @F

@Var @RT(8)cMoveAll @RT(0) @T @F @DT @RT(4)DINT @RT(0) @T @T @BASIC 0 @F
@F @F
@T
@BEG_Attrib
0 @RT(3)100 @RT(32)all movements (for evLockUnlock)
@END_Attrib
1 1 @F @F @F @F

@END_Const

@BEG_Export

@BEG_Kind
@ALGORITHM_BLOCK @RT(13)ABInterpreter @STRUCTURED_TEXT
@RT(0) @RT(0) @RT(0)
@END_Kind

@BEG_Dcl
@RT(16)DclTreeContainer
45
@Var @RT(12)fbLockUnlock @RT(0) @T @T @DERIVED 0 @T @T @DT @RT(12)FBLockUnlock @RT(0) @T @T @UNKNOWN 0 @F
@F @F
@T
@BEG_Attrib
3 @RT(0) @RT(0) @RT(0)
@END_Attrib
1 0 @F @F @F @F

@Var @RT(12)fbDebugTrace @RT(0) @T @T @DERIVED 0 @T @T @DT @RT(12)FBDebugTrace @RT(0) @T @T @UNKNOWN 0 @F
@F @F
@T
@BEG_Attrib
3 @RT(0) @RT(0) @RT(0)
@END_Attrib
1 0 @F @F @F @F

@Var @RT(13)fbDebugTrace2 @RT(0) @T @T @DERIVED 0 @T @T @DT @RT(13)FBDebugTrace2 @RT(0) @T @T @UNKNOWN 0 @F
@F @F
@T
@BEG_Attrib
3 @RT(0) @RT(0) @RT(0)
@END_Attrib
1 0 @F @F @F @F

@Var @RT(14)fbSetStepState @RT(0) @T @T @DERIVED 0 @T @T @DT @RT(14)FBSetStepState @RT(0) @T @T @UNKNOWN 0 @F
@F @F
@T
@BEG_Attrib
3 @RT(0) @RT(0) @RT(0)
@END_Attrib
1 0 @F @F @F @F

@Var @RT(14)sv_ODCSequence @RT(0) @T @T @DERIVED 0 @T @T @DT @RT(13)KODC_Sequence @RT(0) @T @T @UNKNOWN 0 @F
@F @F
@T
@BEG_Attrib
3 @RT(0) @RT(0) @RT(0)
@END_Attrib
1 8 @F @F @F @F

@Var @RT(17)sv_ODCSequenceInt @RT(0) @T @T @DERIVED 0 @T @T @DT @RT(21)tyODCSequenceInternal @RT(0) @T @T @UNKNOWN 0 @F
@F @F
@T
@BEG_Attrib
3 @RT(0) @RT(0) @RT(0)
@END_Attrib
1 8 @F @F @F @F

@Var @RT(21)sv_MovementsAvailable @RT(0) @T @T @DERIVED 0 @T @T @DT @RT(22)tyMovementRegisterList @RT(0) @T @T @UNKNOWN 0 @F
@F @F
@T
@BEG_Attrib
3 @RT(0) @RT(0) @RT(0)
@END_Attrib
1 8 @F @F @F @F

@Var @RT(26)sv_InterpreterParallelInfo @RT(0) @T @T @DERIVED 0 @T @T @DT @RT(17)tyODCParallelInfo @RT(0) @T @T @UNKNOWN 0 @F
@F @F
@T
@BEG_Attrib
3 @RT(0) @RT(0) @RT(0)
@END_Attrib
1 8 @F @F @F @F

@Var @RT(15)evCheckLocklist @RT(0) @T @T @RENAMED 0 @T @T @DT @RT(16)tevCheckLocklist @RT(0) @T @T @UNKNOWN 0 @F
@F @F
@T
@BEG_Attrib
3 @RT(0) @RT(0) @RT(0)
@END_Attrib
1 7 @F @F @F @F

@Var @RT(15)odcParallelInfo @RT(0) @T @T @DERIVED 0 @T @T @DT @RT(17)tyODCParallelInfo @RT(0) @T @T @UNKNOWN 0 @F
@F @F
@T
@BEG_Attrib
3 @RT(0) @RT(0) @RT(0)
@END_Attrib
1 0 @F @F @F @F

@Var @RT(8)miEndRow @RT(0) @T @F @DT @RT(4)DINT @RT(0) @T @T @BASIC 0 @F
@F @F
@T
@BEG_Attrib
3 @RT(0) @RT(25)where ODC stops executing @RT(0)
@END_Attrib
1 0 @F @F @F @F

@Var @RT(5)dummy @RT(0) @T @F @DT @RT(4)DINT @RT(0) @T @T @BASIC 0 @F
@F @F
@T
@BEG_Attrib
3 @RT(0) @RT(0) @RT(0)
@END_Attrib
1 0 @F @F @F @F

@Var @RT(12)mbFatalError @RT(0) @T @F @DT @RT(4)BOOL @RT(0) @T @T @BASIC 0 @F
@F @F
@T
@BEG_Attrib
3 @RT(0) @RT(49)there was some error, interpreting is not allowed @RT(0)
@END_Attrib
1 0 @F @F @F @F

@Var @RT(13)mbNormalError @RT(0) @T @F @DT @RT(4)BOOL @RT(0) @T @T @BASIC 0 @F
@F @F
@T
@BEG_Attrib
3 @RT(0) @RT(49)there was some error, interpreting is not allowed @RT(0)
@END_Attrib
1 0 @F @F @F @F

@Var @RT(8)mbActive @RT(0) @T @F @DT @RT(4)BOOL @RT(0) @T @T @BASIC 0 @F
@F @F
@T
@BEG_Attrib
3 @RT(0) @RT(0) @RT(0)
@END_Attrib
1 0 @F @F @F @F

@Var @RT(10)mbFinished @RT(0) @T @F @DT @RT(4)BOOL @RT(0) @T @T @BASIC 0 @F
@F @F
@T
@BEG_Attrib
3 @RT(0) @RT(0) @RT(0)
@END_Attrib
1 0 @F @F @F @F

@Var @RT(29)sv_StartConditionInstanceData @RT(0) @T @T @DERIVED 0 @T @T @DT @RT(23)tyStartCondInstanceData @RT(0) @T @T @UNKNOWN 0 @F
@F @F
@T
@BEG_Attrib
3 @RT(0) @RT(50)list with start condition params for all instances @RT(0)
@END_Attrib
1 8 @F @F @F @F

@Var @RT(21)sv_ODCDeviceMovements @RT(0) @T @T @DERIVED 0 @T @T @DT @RT(23)tsODCDeviceMovementList @RT(0) @T @T @UNKNOWN 0 @F
@F @F
@T
@BEG_Attrib
3 @RT(0) @RT(0) @RT(0)
@END_Attrib
1 8 @F @F @F @F

@Var @RT(29)sv_CheckConditionInstanceData @RT(0) @T @T @DERIVED 0 @T @T @DT @RT(23)tyCheckCondInstanceData @RT(0) @T @T @UNKNOWN 0 @F
@F @F
@T
@BEG_Attrib
3 @RT(0) @RT(50)list with check condition params for all instances @RT(0)
@END_Attrib
1 8 @F @F @F @F

@Var @RT(22)erMovementNotAvailable @RT(0) @T @F @DT @RT(5)ALARM @RT(0) @T @T @BASIC 0 @F
@F @F
@T
@BEG_Attrib
3 @RT(0) @RT(0) @RT(0)
@END_Attrib
1 7 @F @F @F @F

@Var @RT(18)mCheckCondHelpData @RT(0) @T @T @DERIVED 0 @T @T @DT @RT(19)tyCheckCondHelpData @RT(0) @T @T @UNKNOWN 0 @F
@F @F
@T
@BEG_Attrib
3 @RT(0) @RT(0) @RT(0)
@END_Attrib
1 0 @F @F @F @F

@Var @RT(26)erWaitingForCheckCondition @RT(0) @T @F @DT @RT(5)ALARM @RT(0) @T @T @BASIC 0 @F
@F @F
@T
@BEG_Attrib
3 @RT(0) @RT(0) @RT(0)
@END_Attrib
1 7 @F @F @F @F

@Var @RT(9)sv_bFALSE @RT(0) @T @F @DT @RT(4)BOOL @RT(0) @T @T @BASIC 0 @F
@F @F
@T
@BEG_Attrib
3 @RT(0) @RT(0) @RT(0)
@END_Attrib
1 8 @F @F @F @F

@Var @RT(26)erCompNotInCorrectPosition @RT(0) @T @F @DT @RT(5)ALARM @RT(0) @T @T @BASIC 0 @F
@F @F
@T
@BEG_Attrib
3 @RT(0) @RT(0) @RT(0)
@END_Attrib
1 7 @F @F @F @F

@Var @RT(13)sv_TraceLevel @RT(0) @T @T @DERIVED 0 @F @RT(12)tsTraceLevel @F
@T
@BEG_Attrib
3 @RT(0) @RT(0) @RT(0)
@END_Attrib
1 8 @F @F @F @F

@Var @RT(15)sv_iUsedColumns @RT(0) @T @T @RENAMED 0 @T @T @DT @RT(4)DINT @RT(0) @T @T @BASIC 0 @F
@F @F
@T
@BEG_Attrib
3 @RT(0) @RT(0) @RT(0)
@END_Attrib
1 8 @F @F @F @F

@Var @RT(12)sv_iUsedRows @RT(0) @T @F @DT @RT(4)DINT @RT(0) @T @T @BASIC 0 @F
@F @F
@T
@BEG_Attrib
3 @RT(0) @RT(0) @RT(0)
@END_Attrib
1 8 @F @F @F @F

@Var @RT(16)sv_OperationMode @RT(0) @T @T @DERIVED 0 @T @T @DT @RT(15)tnOperationMode @RT(0) @T @T @UNKNOWN 0 @F
@F @F
@T
@BEG_Attrib
3 @RT(0) @RT(0) @RT(0)
@END_Attrib
1 8 @F @F @F @F

@Var @RT(5)fbRTC @RT(0) @T @T @DERIVED 0 @T @T @DT @RT(3)RTC @RT(0) @T @T @UNKNOWN 0 @F
@F @F
@T
@BEG_Attrib
3 @RT(0) @RT(0) @RT(0)
@END_Attrib
1 0 @F @F @F @F

@Var @RT(29)sv_iDurationUpdateInTolerance @RT(0) @T @F @DT @RT(4)DINT @RT(0) @T @T @BASIC 0 @F
@F @F
@T
@BEG_Attrib
3 @RT(0) @RT(0) @RT(0)
@END_Attrib
1 8 @F @F @F @F

@Var @RT(25)sv_rMoveDurationTolerance @RT(0) @T @F @DT @RT(4)REAL @RT(0) @T @T @BASIC 0 @F
@F @F
@T
@BEG_Attrib
3 @RT(0) @RT(0) @RT(0)
@END_Attrib
1 8 @F @F @F @F

@Var @RT(21)sv_ConditionParameter @RT(0) @T @T @DERIVED 0 @T @T @DT @RT(17)tyIFConditionData @RT(0) @T @T @UNKNOWN 0 @F
@F @F
@T
@BEG_Attrib
3 @RT(0) @RT(0) @RT(0)
@END_Attrib
1 8 @F @F @F @F

@Var @RT(16)sv_LoopParameter @RT(0) @T @T @DERIVED 0 @T @T @DT @RT(10)tyLoopData @RT(0) @T @T @UNKNOWN 0 @F
@F @F
@T
@BEG_Attrib
3 @RT(0) @RT(39)array with data of all programmed loops @RT(0)
@END_Attrib
1 8 @F @F @F @F

@Var @RT(20)mIFConditionHelpData @RT(0) @T @T @DERIVED 0 @T @T @DT @RT(21)tyIFConditionHelpData @RT(0) @T @T @UNKNOWN 0 @F
@F @F
@T
@BEG_Attrib
3 @RT(0) @RT(0) @RT(0)
@END_Attrib
1 0 @F @F @F @F

@Var @RT(13)mLoopHelpData @RT(0) @T @T @DERIVED 0 @T @T @DT @RT(14)tyLoopHelpData @RT(0) @T @T @UNKNOWN 0 @F
@F @F
@T
@BEG_Attrib
3 @RT(0) @RT(0) @RT(0)
@END_Attrib
1 0 @F @F @F @F

@Var @RT(18)sv_GroupActiveData @RT(0) @T @T @DERIVED 0 @T @T @DT @RT(17)tsGroupActiveData @RT(0) @T @T @UNKNOWN 0 @F
@F @F
@T
@BEG_Attrib
3 @RT(0) @RT(0) @RT(0)
@END_Attrib
1 8 @F @F @F @F

@Var @RT(25)g_iAutoCycleLoopStartLine @RT(0) @T @F @DT @RT(4)DINT @RT(0) @T @T @BASIC 0 @F
@F @F
@T
@BEG_Attrib
3 @RT(0) @RT(0) @RT(0)
@END_Attrib
1 6 @F @F @F @F

@Var @RT(23)g_iAutoCycleLoopEndLine @RT(0) @T @F @DT @RT(4)DINT @RT(0) @T @T @BASIC 0 @F
@F @F
@T
@BEG_Attrib
3 @RT(0) @RT(0) @RT(0)
@END_Attrib
1 6 @F @F @F @F

@Var @RT(22)g_ParallelOpenHelpData @RT(0) @T @T @DERIVED 0 @T @T @DT @RT(22)tyParallelOpenHelpData @RT(0) @T @T @UNKNOWN 0 @F
@F @F
@T
@BEG_Attrib
3 @RT(0) @RT(0) @RT(0)
@END_Attrib
1 6 @F @F @F @F

@Var @RT(23)erReadyAndNotPosReached @RT(0) @T @F @DT @RT(5)ALARM @RT(0) @T @T @BASIC 0 @F
@F @F
@T
@BEG_Attrib
3 @RT(0) @RT(0) @RT(0)
@END_Attrib
1 7 @F @F @F @F

@Var @RT(25)sv_StartedManualMovements @RT(0) @T @T @DERIVED 0 @T @T @DT @RT(28)tsStartedMoveDataODCExtended @RT(0) @T @T @UNKNOWN 0 @F
@F @F
@T
@BEG_Attrib
3 @RT(0) @RT(0) @RT(0)
@END_Attrib
1 8 @F @F @F @F

@Var @RT(10)mbStepMode @RT(0) @T @F @DT @RT(4)BOOL @RT(0) @T @T @BASIC 0 @F
@F @F
@T
@BEG_Attrib
3 @RT(0) @RT(0) @RT(0)
@END_Attrib
1 0 @F @F @F @F

@Var @RT(24)erNoStepBwdIntoCondition @RT(0) @T @F @DT @RT(5)ALARM @RT(0) @T @T @BASIC 0 @F
@F @F
@T
@BEG_Attrib
3 @RT(0) @RT(0) @RT(0)
@END_Attrib
1 7 @F @F @F @F

@Var @RT(19)erNoStepBwdIntoLoop @RT(0) @T @F @DT @RT(5)ALARM @RT(0) @T @T @BASIC 0 @F
@F @F
@T
@BEG_Attrib
3 @RT(0) @RT(0) @RT(0)
@END_Attrib
1 7 @F @F @F @F

@Var @RT(20)erNoStepBwdOutOfLoop @RT(0) @T @F @DT @RT(5)ALARM @RT(0) @T @T @BASIC 0 @F
@F @F
@T
@BEG_Attrib
3 @RT(0) @RT(0) @RT(0)
@END_Attrib
1 7 @F @F @F @F

@END_Dcl

@END_Export

@BEG_Body

38

@BEG_Export

@BEG_Algo
@ALGORITHM @RT(16)aCorrectDuration @STRUCTURED_TEXT
@RT(0) @RT(0) @RT(0) @F @F
@END_Algo

@BEG_Dcl
@RT(16)DclTreeContainer
11
@Var @RT(9)pMoveData @RT(0) @T @T @REFTO 0 @F @DERIVED 0 @T @T @DT @RT(10)tsMoveData @RT(0) @T @T @UNKNOWN 0 @F
@F @F
@T
@BEG_Attrib
3 @RT(0) @RT(0) @RT(0)
@END_Attrib
1 2 @F @F @F @F

@Var @RT(7)iColumn @RT(0) @T @F @DT @RT(4)DINT @RT(0) @T @T @BASIC 0 @F
@F @F
@T
@BEG_Attrib
3 @RT(0) @RT(0) @RT(0)
@END_Attrib
1 1 @F @F @F @F

@Var @RT(9)dDuration @RT(0) @T @F @DT @RT(4)TIME @RT(0) @T @T @BASIC 0 @F
@F @F
@T
@BEG_Attrib
3 @RT(0) @RT(0) @RT(0)
@END_Attrib
1 0 @F @F @F @F

@Var @RT(8)dActTime @RT(0) @T @F @DT @RT(13)DATE_AND_TIME @RT(0) @T @T @BASIC 0 @F
@F @F
@T
@BEG_Attrib
3 @RT(0) @RT(0) @RT(0)
@END_Attrib
1 0 @F @F @F @F

@Var @RT(14)dMovementDelay @RT(0) @T @F @DT @RT(4)TIME @RT(0) @T @T @BASIC 0 @F
@F @F
@T
@BEG_Attrib
3 @RT(0) @RT(0) @RT(0)
@END_Attrib
1 0 @F @F @F @F

@Var @RT(8)DeviceId @RT(0) @T @T @DERIVED 0 @T @T @DT @RT(10)tsDeviceId @RT(0) @T @T @UNKNOWN 0 @F
@F @F
@T
@BEG_Attrib
3 @RT(0) @RT(0) @RT(0)
@END_Attrib
1 1 @F @F @F @F

@Var @RT(5)rTmp1 @RT(0) @T @F @DT @RT(4)REAL @RT(0) @T @T @BASIC 0 @F
@F @F
@T
@BEG_Attrib
3 @RT(0) @RT(0) @RT(0)
@END_Attrib
1 0 @F @F @F @F

@Var @RT(5)rTmp2 @RT(0) @T @F @DT @RT(4)REAL @RT(0) @T @T @BASIC 0 @F
@F @F
@T
@BEG_Attrib
3 @RT(0) @RT(0) @RT(0)
@END_Attrib
1 0 @F @F @F @F

@Var @RT(18)fbUpdateProperties @RT(0) @T @T @DERIVED 0 @T @T @DT @RT(24)FBUpdateEditorProperties @RT(0) @T @T @UNKNOWN 0 @F
@F @F
@T
@BEG_Attrib
3 @RT(0) @RT(0) @RT(0)
@END_Attrib
1 0 @F @F @F @F

@Var @RT(9)bInitDone @RT(0) @T @F @DT @RT(4)BOOL @RT(0) @T @T @BASIC 0 @F
@F @F
@T
@BEG_Attrib
3 @RT(0) @RT(0) @RT(0)
@END_Attrib
1 0 @F @F @F @F

@Var @RT(10)dCycleTime @RT(0) @T @F @DT @RT(4)TIME @RT(0) @T @T @BASIC 0 @F
@F @F
@T
@BEG_Attrib
3 @RT(0) @RT(0) @RT(0)
@END_Attrib
1 0 @F @F @F @F

@END_Dcl

@END_Export

@BEG_Export

@BEG_Algo
@ALGORITHM @RT(21)aCheckConditionUnlock @STRUCTURED_TEXT
@RT(0) @RT(0) @RT(0) @F @F
@END_Algo

@BEG_Dcl
@RT(16)DclTreeContainer
1
@Var @RT(1)i @RT(0) @T @F @DT @RT(4)DINT @RT(0) @T @T @BASIC 0 @F
@F @F
@T
@BEG_Attrib
3 @RT(0) @RT(0) @RT(0)
@END_Attrib
1 4 @F @F @F @F

@END_Dcl

@END_Export

@BEG_Export

@BEG_Algo
@ALGORITHM @RT(17)aResetInterpreter @STRUCTURED_TEXT
@RT(0) @RT(0) @RT(0) @F @F
@END_Algo

@BEG_Dcl
@RT(16)DclTreeContainer
2
@Var @RT(1)i @RT(0) @T @F @DT @RT(4)DINT @RT(0) @T @T @BASIC 0 @F
@F @F
@T
@BEG_Attrib
3 @RT(0) @RT(0) @RT(0)
@END_Attrib
1 4 @F @F @F @F

@Var @RT(21)bExcludeActiveColumns @RT(0) @T @F @DT @RT(4)BOOL @RT(0) @T @T @BASIC 0 @F
@F @F
@T
@BEG_Attrib
3 @RT(0) @RT(67)TRUE: do not reset active columns (possible with StartParallelOpen) @RT(0)
@END_Attrib
1 1 @F @F @F @F

@END_Dcl

@END_Export

@BEG_Export

@BEG_Algo
@ALGORITHM @RT(24)aStopInterpreterInternal @STRUCTURED_TEXT
@RT(0) @RT(0) @RT(0) @F @F
@END_Algo

@BEG_Dcl
@RT(16)DclTreeContainer
5
@Var @RT(12)bNormalError @RT(0) @T @F @DT @RT(4)BOOL @RT(0) @T @T @BASIC 0 @F
@F @F
@T
@BEG_Attrib
3 @RT(0) @RT(0) @RT(0)
@END_Attrib
1 1 @F @F @F @F

@Var @RT(11)bFatalError @RT(0) @T @F @DT @RT(4)BOOL @RT(0) @T @T @BASIC 0 @F
@F @F
@T
@BEG_Attrib
3 @RT(0) @RT(0) @RT(0)
@END_Attrib
1 1 @F @F @F @F

@Var @RT(22)fbStopStartedMovements @RT(0) @T @T @DERIVED 0 @T @T @DT @RT(22)FBStopStartedMovements @RT(0) @T @T @UNKNOWN 0 @F
@F @F
@T
@BEG_Attrib
3 @RT(0) @RT(0) @RT(0)
@END_Attrib
1 0 @F @F @F @F

@Var @RT(28)fbStopStartedManualMovements @RT(0) @T @T @DERIVED 0 @T @T @DT @RT(28)FBStopStartedManualMovements @RT(0) @T @T @UNKNOWN 0 @F
@F @F
@T
@BEG_Attrib
3 @RT(0) @RT(0) @RT(0)
@END_Attrib
1 0 @F @F @F @F

@Var @RT(11)DeviceIdAll @RT(0) @T @T @DERIVED 0 @T @T @DT @RT(10)tsDeviceId @RT(0) @T @T @UNKNOWN 0 @F
@F @F
@T
@BEG_Attrib
3 @RT(0) @RT(0) @RT(0)
@END_Attrib
1 0 @F @F @F @F

@END_Dcl

@END_Export

@BEG_Export

@BEG_Algo
@ALGORITHM @RT(21)aStopInterpreterFatal @STRUCTURED_TEXT
@RT(0) @RT(0) @RT(0) @F @F
@END_Algo

@BEG_Dcl
@RT(16)DclTreeContainer
0
@END_Dcl

@END_Export

@BEG_Export

@BEG_Algo
@ALGORITHM @RT(15)aCheckActivated @STRUCTURED_TEXT
@RT(0) @RT(0) @RT(0) @F @F
@END_Algo

@BEG_Dcl
@RT(16)DclTreeContainer
4
@Var @RT(8)DeviceId @RT(0) @T @T @DERIVED 0 @T @T @DT @RT(10)tsDeviceId @RT(0) @T @T @UNKNOWN 0 @F
@F @F
@T
@BEG_Attrib
3 @RT(0) @RT(0) @RT(0)
@END_Attrib
1 1 @F @F @F @F

@Var @RT(8)MoveData @RT(0) @T @T @DERIVED 0 @T @T @DT @RT(10)tsMoveData @RT(0) @T @T @UNKNOWN 0 @F
@F @F
@T
@BEG_Attrib
3 @RT(0) @RT(0) @RT(0)
@END_Attrib
1 1 @F @F @F @F

@Var @RT(10)bActivated @RT(0) @T @F @DT @RT(4)BOOL @RT(0) @T @T @BASIC 0 @F
@F @F
@T
@BEG_Attrib
3 @RT(0) @RT(0) @RT(0)
@END_Attrib
1 3 @F @F @F @F

@Var @RT(8)iFuIndex @RT(0) @T @F @DT @RT(4)DINT @RT(0) @T @T @BASIC 0 @F
@F @F
@T
@BEG_Attrib
3 @RT(0) @RT(0) @RT(0)
@END_Attrib
1 4 @F @F @F @F

@END_Dcl

@END_Export

@BEG_Export

@BEG_Algo
@ALGORITHM @RT(12)aIncreaseRow @STRUCTURED_TEXT
@RT(0) @RT(0) @RT(0) @F @F
@END_Algo

@BEG_Dcl
@RT(16)DclTreeContainer
8
@Var @RT(7)iColumn @RT(0) @T @F @DT @RT(4)DINT @RT(0) @T @T @BASIC 0 @F
@F @F
@T
@BEG_Attrib
3 @RT(0) @RT(0) @RT(0)
@END_Attrib
1 1 @F @F @F @F

@Var @RT(8)iTmpLine @RT(0) @T @F @DT @RT(4)DINT @RT(0) @T @T @BASIC 0 @F
@F @F
@T
@BEG_Attrib
3 @RT(0) @RT(0) @RT(0)
@END_Attrib
1 4 @F @F @F @F

@Var @RT(7)iEndRow @RT(0) @T @F @DT @RT(4)DINT @RT(0) @T @T @BASIC 0 @F
@F @F
@T
@BEG_Attrib
3 @RT(0) @RT(0) @RT(0)
@END_Attrib
1 1 @F @F @F @F

@Var @RT(22)iStopEverythingCounter @RT(0) @T @F @DT @RT(4)DINT @RT(0) @T @T @BASIC 0 @F
@F @F
@T
@BEG_Attrib
3 @RT(0) @RT(0) @RT(0)
@END_Attrib
1 0 @F @F @F @F

@Var @RT(1)k @RT(0) @T @F @DT @RT(4)DINT @RT(0) @T @T @BASIC 0 @F
@F @F
@T
@BEG_Attrib
3 @RT(0) @RT(0) @RT(0)
@END_Attrib
1 4 @F @F @F @F

@Var @RT(6)iCount @RT(0) @T @F @DT @RT(3)INT @RT(0) @T @T @BASIC 0 @F
@F @F
@T
@BEG_Attrib
3 @RT(0) @RT(0) @RT(0)
@END_Attrib
1 0 @F @F @F @F

@Var @RT(14)fbSetStepState @RT(0) @T @T @DERIVED 0 @T @T @DT @RT(14)FBSetStepState @RT(0) @T @T @UNKNOWN 0 @F
@F @F
@T
@BEG_Attrib
3 @RT(0) @RT(0) @RT(0)
@END_Attrib
1 0 @F @F @F @F

@Var @RT(9)pMoveData @RT(0) @T @T @REFTO 0 @F @DERIVED 0 @T @T @DT @RT(10)tsMoveData @RT(0) @T @T @UNKNOWN 0 @F
@F @F
@T
@BEG_Attrib
3 @RT(0) @RT(0) @RT(0)
@END_Attrib
1 0 @F @F @F @F

@END_Dcl

@END_Export

@BEG_Export

@BEG_Algo
@ALGORITHM @RT(19)aFindCheckCondition @STRUCTURED_TEXT
@RT(0) @RT(0) @RT(0) @F @F
@END_Algo

@BEG_Dcl
@RT(16)DclTreeContainer
3
@Var @RT(1)i @RT(0) @T @F @DT @RT(4)DINT @RT(0) @T @T @BASIC 0 @F
@F @F
@T
@BEG_Attrib
3 @RT(0) @RT(0) @RT(0)
@END_Attrib
1 4 @F @F @F @F

@Var @RT(8)Movement @RT(0) @T @T @DERIVED 0 @T @T @DT @RT(9)KODC_Step @RT(0) @T @T @UNKNOWN 0 @F
@F @F
@T
@BEG_Attrib
3 @RT(0) @RT(18)requested movement @RT(0)
@END_Attrib
1 1 @F @F @F @F

@Var @RT(6)bFound @RT(0) @T @F @DT @RT(4)BOOL @RT(0) @T @T @BASIC 0 @F
@F @F
@T
@BEG_Attrib
3 @RT(0) @RT(44)check condition for requested movement found @RT(0)
@END_Attrib
1 3 @F @F @F @F

@END_Dcl

@END_Export

@BEG_Export

@BEG_Algo
@ALGORITHM @RT(21)aStopInterpreterError @STRUCTURED_TEXT
@RT(0) @RT(0) @RT(0) @F @F
@END_Algo

@BEG_Dcl
@RT(16)DclTreeContainer
0
@END_Dcl

@END_Export

@BEG_Export

@BEG_Algo
@ALGORITHM @RT(22)aStopInterpreterNormal @STRUCTURED_TEXT
@RT(0) @RT(0) @RT(0) @F @F
@END_Algo

@BEG_Dcl
@RT(16)DclTreeContainer
0
@END_Dcl

@END_Export

@BEG_Export

@BEG_Algo
@ALGORITHM @RT(20)aCheckSequenceSanity @STRUCTURED_TEXT
@RT(0) @RT(0) @RT(0) @F @F
@END_Algo

@BEG_Dcl
@RT(16)DclTreeContainer
8
@Var @RT(3)bOK @RT(0) @T @F @DT @RT(4)BOOL @RT(0) @T @T @BASIC 0 @F
@F @F
@T
@BEG_Attrib
3 @RT(0) @RT(20)Sanity checks passed @RT(0)
@END_Attrib
1 3 @F @F @F @F

@Var @RT(7)iColumn @RT(0) @T @F @DT @RT(4)DINT @RT(0) @T @T @BASIC 0 @F
@F @F
@T
@BEG_Attrib
3 @RT(0) @RT(0) @RT(0)
@END_Attrib
1 4 @F @F @F @F

@Var @RT(4)iRow @RT(0) @T @F @DT @RT(4)DINT @RT(0) @T @T @BASIC 0 @F
@F @F
@T
@BEG_Attrib
3 @RT(0) @RT(0) @RT(0)
@END_Attrib
1 4 @F @F @F @F

@Var @RT(17)iEndParallelFound @RT(0) @T @F @DT @RT(4)DINT @RT(0) @T @T @BASIC 0 @F
@F @F
@T
@BEG_Attrib
3 @RT(0) @RT(0) @RT(0)
@END_Attrib
1 4 @F @F @F @F

@Var @RT(19)iStartParallelFound @RT(0) @T @F @DT @RT(4)DINT @RT(0) @T @T @BASIC 0 @F
@F @F
@T
@BEG_Attrib
3 @RT(0) @RT(0) @RT(0)
@END_Attrib
1 4 @F @F @F @F

@Var @RT(19)bAutoCycleLoopFound @RT(0) @T @F @DT @RT(4)BOOL @RT(0) @T @T @BASIC 0 @F
@F @F
@T
@BEG_Attrib
3 @RT(0) @RT(32)autocycle loop found in sequence @RT(0)
@END_Attrib
1 3 @F @F @F @F

@Var @RT(15)iEndSequenceRow @RT(0) @T @F @DT @RT(4)DINT @RT(0) @T @T @BASIC 0 @F
@F @F
@T
@BEG_Attrib
3 @RT(0) @RT(43)line number where ODC.EndSequence was found @RT(0)
@END_Attrib
1 3 @F @F @F @F

@Var @RT(18)iNoOfStartParallel @RT(0) @T @F @DT @RT(4)DINT @RT(0) @T @T @BASIC 0 @F
@F @F
@T
@BEG_Attrib
3 @RT(0) @RT(47)number of "StartParallel" steps in the sequence @RT(0)
@END_Attrib
1 3 @F @F @F @F

@END_Dcl

@END_Export

@BEG_Export

@BEG_Algo
@ALGORITHM @RT(22)aClearInternalSequence @STRUCTURED_TEXT
@RT(0) @RT(0) @RT(0) @F @F
@END_Algo

@BEG_Dcl
@RT(16)DclTreeContainer
5
@Var @RT(7)iColumn @RT(0) @T @F @DT @RT(4)DINT @RT(0) @T @T @BASIC 0 @F
@F @F
@T
@BEG_Attrib
3 @RT(0) @RT(0) @RT(0)
@END_Attrib
1 4 @F @F @F @F

@Var @RT(4)iRow @RT(0) @T @F @DT @RT(4)DINT @RT(0) @T @T @BASIC 0 @F
@F @F
@T
@BEG_Attrib
3 @RT(0) @RT(0) @RT(0)
@END_Attrib
1 4 @F @F @F @F

@Var @RT(9)EmptyStep @RT(0) @T @T @DERIVED 0 @T @T @DT @RT(17)tsODCStepInternal @RT(0) @T @T @UNKNOWN 0 @F
@F @F
@T
@BEG_Attrib
3 @RT(0) @RT(0) @RT(0)
@END_Attrib
1 0 @F @F @F @F

@Var @RT(1)i @RT(0) @T @F @DT @RT(4)DINT @RT(0) @T @T @BASIC 0 @F
@F @F
@T
@BEG_Attrib
3 @RT(0) @RT(0) @RT(0)
@END_Attrib
1 4 @F @F @F @F

@Var @RT(15)EmptyDependency @RT(0) @T @T @DERIVED 0 @T @T @DT @RT(20)tyODCDependencyArray @RT(0) @T @T @UNKNOWN 0 @F
@F @F
@T
@BEG_Attrib
3 @RT(0) @RT(0) @RT(0)
@END_Attrib
1 0 @F @F @F @F

@END_Dcl

@END_Export

@BEG_Export

@BEG_Algo
@ALGORITHM @RT(16)aGetMovementData @STRUCTURED_TEXT
@RT(0) @RT(0) @RT(0) @F @F
@END_Algo

@BEG_Dcl
@RT(16)DclTreeContainer
7
@Var @RT(8)Movement @RT(0) @T @T @DERIVED 0 @T @T @DT @RT(9)KODC_Step @RT(0) @T @T @UNKNOWN 0 @F
@F @F
@T
@BEG_Attrib
3 @RT(0) @RT(0) @RT(0)
@END_Attrib
1 1 @F @F @F @F

@Var @RT(9)Direction @RT(0) @T @T @DERIVED 0 @T @T @DT @RT(15)tnMoveDirection @RT(0) @T @T @UNKNOWN 0 @F
@F @F
@T
@BEG_Attrib
3 @RT(0) @RT(38)movedirection (min to max, max to min) @RT(0)
@END_Attrib
1 3 @F @F @F @F

@Var @RT(10)prActValue @RT(0) @T @T @REFTO 0 @T @DT @RT(4)REAL @RT(0) @T @T @BASIC 0 @F
@F @F
@T
@BEG_Attrib
3 @RT(0) @RT(35)refto actual value of this movement @RT(0)
@END_Attrib
1 3 @F @F @F @F

@Var @RT(20)pbReferenceCondition @RT(0) @T @T @REFTO 0 @T @DT @RT(4)BOOL @RT(0) @T @T @BASIC 0 @F
@F @F
@T
@BEG_Attrib
3 @RT(0) @RT(35)refto actual value of this movement @RT(0)
@END_Attrib
1 3 @F @F @F @F

@Var @RT(8)DeviceId @RT(0) @T @T @DERIVED 0 @T @T @DT @RT(10)tsDeviceId @RT(0) @T @T @UNKNOWN 0 @F
@F @F
@T
@BEG_Attrib
3 @RT(0) @RT(0) @RT(0)
@END_Attrib
1 0 @F @F @F @F

@Var @RT(1)i @RT(0) @T @F @DT @RT(4)DINT @RT(0) @T @T @BASIC 0 @F
@F @F
@T
@BEG_Attrib
3 @RT(0) @RT(0) @RT(0)
@END_Attrib
1 4 @F @F @F @F

@Var @RT(1)k @RT(0) @T @F @DT @RT(4)DINT @RT(0) @T @T @BASIC 0 @F
@F @F
@T
@BEG_Attrib
3 @RT(0) @RT(0) @RT(0)
@END_Attrib
1 4 @F @F @F @F

@END_Dcl

@END_Export

@BEG_Export

@BEG_Algo
@ALGORITHM @RT(18)aGetLockUnlockData @STRUCTURED_TEXT
@RT(0) @RT(0) @RT(0) @F @F
@END_Algo

@BEG_Dcl
@RT(16)DclTreeContainer
1
@Var @RT(9)iInstance @RT(0) @T @F @DT @RT(4)DINT @RT(0) @T @T @BASIC 0 @F
@F @F
@T
@BEG_Attrib
3 @RT(0) @RT(0) @RT(0)
@END_Attrib
1 1 @F @F @F @F

@END_Dcl

@END_Export

@BEG_Export

@BEG_Algo
@ALGORITHM @RT(27)aInitCheckConditionHelpData @STRUCTURED_TEXT
@RT(0) @RT(0) @RT(0) @F @F
@END_Algo

@BEG_Dcl
@RT(16)DclTreeContainer
3
@Var @RT(8)DeviceId @RT(0) @T @T @DERIVED 0 @T @T @DT @RT(10)tsDeviceId @RT(0) @T @T @UNKNOWN 0 @F
@F @F
@T
@BEG_Attrib
3 @RT(0) @RT(0) @RT(0)
@END_Attrib
1 0 @F @F @F @F

@Var @RT(17)fbCheckPosReached @RT(0) @T @T @DERIVED 0 @T @T @DT @RT(17)FBCheckPosReached @RT(0) @T @T @UNKNOWN 0 @F
@F @F
@T
@BEG_Attrib
3 @RT(0) @RT(0) @RT(0)
@END_Attrib
1 0 @F @F @F @F

@Var @RT(1)i @RT(0) @T @F @DT @RT(4)DINT @RT(0) @T @T @BASIC 0 @F
@F @F
@T
@BEG_Attrib
3 @RT(0) @RT(0) @RT(0)
@END_Attrib
1 4 @F @F @F @F

@END_Dcl

@END_Export

@BEG_Export

@BEG_Algo
@ALGORITHM @RT(24)aInitIFConditionHelpData @STRUCTURED_TEXT
@RT(0) @RT(0) @RT(0) @F @F
@END_Algo

@BEG_Dcl
@RT(16)DclTreeContainer
2
@Var @RT(1)i @RT(0) @T @F @DT @RT(4)DINT @RT(0) @T @T @BASIC 0 @F
@F @F
@T
@BEG_Attrib
3 @RT(0) @RT(0) @RT(0)
@END_Attrib
1 4 @F @F @F @F

@Var @RT(5)state @RT(0) @T @T @DERIVED 0 @T @T @DT @RT(11)KSYS_Status @RT(0) @T @T @UNKNOWN 0 @F
@F @F
@T
@BEG_Attrib
3 @RT(0) @RT(0) @RT(0)
@END_Attrib
1 0 @F @F @F @F

@END_Dcl

@END_Export

@BEG_Export

@BEG_Algo
@ALGORITHM @RT(17)aInitLoopHelpData @STRUCTURED_TEXT
@RT(0) @RT(0) @RT(0) @F @F
@END_Algo

@BEG_Dcl
@RT(16)DclTreeContainer
2
@Var @RT(1)i @RT(0) @T @F @DT @RT(4)DINT @RT(0) @T @T @BASIC 0 @F
@F @F
@T
@BEG_Attrib
3 @RT(0) @RT(0) @RT(0)
@END_Attrib
1 4 @F @F @F @F

@Var @RT(5)state @RT(0) @T @T @DERIVED 0 @T @T @DT @RT(11)KSYS_Status @RT(0) @T @T @UNKNOWN 0 @F
@F @F
@T
@BEG_Attrib
3 @RT(0) @RT(0) @RT(0)
@END_Attrib
1 0 @F @F @F @F

@END_Dcl

@END_Export

@BEG_Export

@BEG_Algo
@ALGORITHM @RT(23)aCreateInternalSequence @STRUCTURED_TEXT
@RT(0) @RT(0) @RT(0) @F @F
@END_Algo

@BEG_Dcl
@RT(16)DclTreeContainer
20
@Var @RT(6)bError @RT(0) @T @F @DT @RT(4)BOOL @RT(0) @T @T @BASIC 0 @F
@F @F
@T
@BEG_Attrib
3 @RT(0) @RT(0) @RT(0)
@END_Attrib
1 3 @F @F @F @F

@Var @RT(12)iUsedColumns @RT(0) @T @F @DT @RT(4)DINT @RT(0) @T @T @BASIC 0 @F
@F @F
@T
@BEG_Attrib
3 @RT(0) @RT(31)maximum usage of sequence array @RT(0)
@END_Attrib
1 3 @F @F @F @F

@Var @RT(9)iUsedRows @RT(0) @T @F @DT @RT(4)DINT @RT(0) @T @T @BASIC 0 @F
@F @F
@T
@BEG_Attrib
3 @RT(0) @RT(31)maximum usage of sequence array @RT(0)
@END_Attrib
1 3 @F @F @F @F

@Var @RT(30)fbInterpreterFindEndOfParallel @RT(0) @T @T @DERIVED 0 @T @T @DT @RT(30)FBInterpreterFindEndOfParallel @RT(0) @T @T @UNKNOWN 0 @F
@F @F
@T
@BEG_Attrib
3 @RT(0) @RT(0) @RT(0)
@END_Attrib
1 0 @F @F @F @F

@Var @RT(15)fbGetMoveNumber @RT(0) @T @T @DERIVED 0 @T @T @DT @RT(15)FBGetMoveNumber @RT(0) @T @T @UNKNOWN 0 @F
@F @F
@T
@BEG_Attrib
3 @RT(0) @RT(0) @RT(0)
@END_Attrib
1 0 @F @F @F @F

@Var @RT(10)ParseStack @RT(0) @T @T @DERIVED 0 @T @T @DT @RT(18)tyNumberParseArray @RT(0) @T @T @UNKNOWN 0 @F
@F @F
@T
@BEG_Attrib
3 @RT(0) @RT(0) @RT(0)
@END_Attrib
1 0 @F @F @F @F

@Var @RT(15)CurrentParsePos @RT(0) @T @T @DERIVED 0 @T @T @DT @RT(20)tsNumberParseElement @RT(0) @T @T @UNKNOWN 0 @F
@F @F
@T
@BEG_Attrib
3 @RT(0) @RT(0) @RT(0)
@END_Attrib
1 0 @F @F @F @F

@Var @RT(7)PrevPos @RT(0) @T @T @DERIVED 0 @T @T @DT @RT(12)tsODCStepPos @RT(0) @T @T @UNKNOWN 0 @F
@F @F
@T
@BEG_Attrib
3 @RT(0) @RT(46)remember prev step for filling out PosPrevStep @RT(0)
@END_Attrib
1 0 @F @F @F @F

@Var @RT(8)iCounter @RT(0) @T @F @DT @RT(4)DINT @RT(0) @T @T @BASIC 0 @F
@F @F
@T
@BEG_Attrib
3 @RT(0) @RT(32)counter for sequential numbering @RT(0)
@END_Attrib
1 0 @F @F @F @F

@Var @RT(18)iParseStackPointer @RT(0) @T @F @DT @RT(4)DINT @RT(0) @T @T @BASIC 0 @F
@F @F
@T
@BEG_Attrib
3 @RT(0) @RT(0) @RT(0)
@END_Attrib
1 0 @F @F @F @F

@Var @RT(8)bEndLoop @RT(0) @T @F @DT @RT(4)BOOL @RT(0) @T @T @BASIC 0 @F
@F @F
@T
@BEG_Attrib
3 @RT(0) @RT(18)end numbering loop @RT(0)
@END_Attrib
1 0 @F @F @F @F

@Var @RT(16)bAddPrevNextInfo @RT(0) @T @F @DT @RT(4)BOOL @RT(0) @T @T @BASIC 0 @F
@F @F
@T
@BEG_Attrib
3 @RT(0) @RT(53)write PosNextStep PosPrevStep variables for this step @RT(0)
@END_Attrib
1 0 @F @F @F @F

@Var @RT(1)m @RT(0) @T @F @DT @RT(4)DINT @RT(0) @T @T @BASIC 0 @F
@F @F
@T
@BEG_Attrib
3 @RT(0) @RT(0) @RT(0)
@END_Attrib
1 4 @F @F @F @F

@Var @RT(1)k @RT(0) @T @F @DT @RT(4)DINT @RT(0) @T @T @BASIC 0 @F
@F @F
@T
@BEG_Attrib
3 @RT(0) @RT(0) @RT(0)
@END_Attrib
1 4 @F @F @F @F

@Var @RT(7)iTmpCol @RT(0) @T @F @DT @RT(4)DINT @RT(0) @T @T @BASIC 0 @F
@F @F
@T
@BEG_Attrib
3 @RT(0) @RT(0) @RT(0)
@END_Attrib
1 4 @F @F @F @F

@Var @RT(11)CurrentStep @RT(0) @T @T @DERIVED 0 @T @T @DT @RT(9)KODC_Step @RT(0) @T @T @UNKNOWN 0 @F
@F @F
@T
@BEG_Attrib
3 @RT(0) @RT(0) @RT(0)
@END_Attrib
1 0 @F @F @F @F

@Var @RT(8)bChanged @RT(0) @T @F @DT @RT(4)BOOL @RT(0) @T @T @BASIC 0 @F
@F @F
@T
@BEG_Attrib
3 @RT(0) @RT(49)need to write back changed step to sv_ODCSequence @RT(0)
@END_Attrib
1 4 @F @F @F @F

@Var @RT(12)bInvalidStep @RT(0) @T @F @DT @RT(4)BOOL @RT(0) @T @T @BASIC 0 @F
@F @F
@T
@BEG_Attrib
3 @RT(0) @RT(58)step is invalid because i has a strange movement/device ID @RT(0)
@END_Attrib
1 4 @F @F @F @F

@Var @RT(23)bContinueAfterLoopAdded @RT(0) @T @F @DT @RT(4)BOOL @RT(0) @T @T @BASIC 0 @F
@F @F
@T
@BEG_Attrib
3 @RT(0) @RT(0) @RT(0)
@END_Attrib
1 0 @F @F @F @F

@Var @RT(14)fbSetStepState @RT(0) @T @T @DERIVED 0 @T @T @DT @RT(14)FBSetStepState @RT(0) @T @T @UNKNOWN 0 @F
@F @F
@T
@BEG_Attrib
3 @RT(0) @RT(0) @RT(0)
@END_Attrib
1 0 @F @F @F @F

@END_Dcl

@END_Export

@BEG_Export

@BEG_Algo
@ALGORITHM @RT(25)aAddStartedManualMovement @STRUCTURED_TEXT
@RT(0) @RT(0) @RT(0) @F @F
@END_Algo

@BEG_Dcl
@RT(16)DclTreeContainer
7
@Var @RT(8)DeviceId @RT(0) @T @T @DERIVED 0 @T @T @DT @RT(10)tsDeviceId @RT(0) @T @T @UNKNOWN 0 @F
@F @F
@T
@BEG_Attrib
3 @RT(0) @RT(0) @RT(0)
@END_Attrib
1 1 @F @F @F @F

@Var @RT(7)StepPos @RT(0) @T @T @DERIVED 0 @T @T @DT @RT(12)tsODCStepPos @RT(0) @T @T @UNKNOWN 0 @F
@F @F
@T
@BEG_Attrib
3 @RT(0) @RT(0) @RT(0)
@END_Attrib
1 1 @F @F @F @F

@Var @RT(6)MoveId @RT(0) @T @T @DERIVED 0 @T @T @DT @RT(10)tMoveIdent @RT(0) @T @T @UNKNOWN 0 @F
@F @F
@T
@BEG_Attrib
3 @RT(0) @RT(0) @RT(0)
@END_Attrib
1 1 @F @F @F @F

@Var @RT(7)MoveDir @RT(0) @T @T @DERIVED 0 @T @T @DT @RT(10)tMoveIdent @RT(0) @T @T @UNKNOWN 0 @F
@F @F
@T
@BEG_Attrib
3 @RT(0) @RT(0) @RT(0)
@END_Attrib
1 1 @F @F @F @F

@Var @RT(9)iInstance @RT(0) @T @F @DT @RT(4)DINT @RT(0) @T @T @BASIC 0 @F
@F @F
@T
@BEG_Attrib
3 @RT(0) @RT(0) @RT(0)
@END_Attrib
1 1 @F @F @F @F

@Var @RT(3)bOK @RT(0) @T @F @DT @RT(4)BOOL @RT(0) @T @T @BASIC 0 @F
@F @F
@T
@BEG_Attrib
3 @RT(0) @RT(0) @RT(0)
@END_Attrib
1 3 @F @F @F @F

@Var @RT(22)fbStartedMovementAdder @RT(0) @T @T @DERIVED 0 @T @T @DT @RT(22)FBStartedMovementAdder @RT(0) @T @T @UNKNOWN 0 @F
@F @F
@T
@BEG_Attrib
3 @RT(0) @RT(0) @RT(0)
@END_Attrib
1 0 @F @F @F @F

@END_Dcl

@END_Export

@BEG_Export

@BEG_Algo
@ALGORITHM @RT(16)aInitInterpreter @STRUCTURED_TEXT
@RT(0) @RT(0) @RT(0) @F @F
@END_Algo

@BEG_Dcl
@RT(16)DclTreeContainer
5
@Var @RT(7)iColumn @RT(0) @T @F @DT @RT(4)DINT @RT(0) @T @T @BASIC 0 @F
@F @F
@T
@BEG_Attrib
3 @RT(0) @RT(31)Column where to start execution @RT(0)
@END_Attrib
1 1 @F @F @F @F

@Var @RT(4)iRow @RT(0) @T @F @DT @RT(4)DINT @RT(0) @T @T @BASIC 0 @F
@F @F
@T
@BEG_Attrib
3 @RT(0) @RT(28)Row where to start execution @RT(0)
@END_Attrib
1 1 @F @F @F @F

@Var @RT(7)iEndRow @RT(0) @T @F @DT @RT(4)DINT @RT(0) @T @T @BASIC 0 @F
@F @F
@T
@BEG_Attrib
3 @RT(0) @RT(30)Column where to stop execution @RT(0)
@END_Attrib
1 1 @F @F @F @F

@Var @RT(22)bSkipAlreadyPosReached @RT(0) @T @F @DT @RT(4)BOOL @RT(0) @T @T @BASIC 0 @F
@F @F
@T
@BEG_Attrib
3 @RT(0) @RT(73)Do not start movements wher PosReached is already TRUE before starting it @RT(0)
@END_Attrib
1 1 @F @F @F @F

@Var @RT(21)bExcludeActiveColumns @RT(0) @T @F @DT @RT(4)BOOL @RT(0) @T @T @BASIC 0 @F
@F @F
@T
@BEG_Attrib
3 @RT(0) @RT(34)do not reset / init active columns @RT(0)
@END_Attrib
1 1 @F @F @F @F

@END_Dcl

@END_Export

@BEG_Export

@BEG_Algo
@ALGORITHM @RT(22)aCheckConditionsManual @STRUCTURED_TEXT
@RT(0) @RT(0) @RT(0) @F @F
@END_Algo

@BEG_Dcl
@RT(16)DclTreeContainer
7
@Var @RT(1)i @RT(0) @T @F @DT @RT(4)DINT @RT(0) @T @T @BASIC 0 @F
@F @F
@T
@BEG_Attrib
3 @RT(0) @RT(0) @RT(0)
@END_Attrib
1 4 @F @F @F @F

@Var @RT(8)Movement @RT(0) @T @T @DERIVED 0 @T @T @DT @RT(9)KODC_Step @RT(0) @T @T @UNKNOWN 0 @F
@F @F
@T
@BEG_Attrib
3 @RT(0) @RT(18)requested movement @RT(0)
@END_Attrib
1 1 @F @F @F @F

@Var @RT(19)bTargetValueReached @RT(0) @T @F @DT @RT(4)BOOL @RT(0) @T @T @BASIC 0 @F
@F @F
@T
@BEG_Attrib
3 @RT(0) @RT(0) @RT(0)
@END_Attrib
1 0 @F @F @F @F

@Var @RT(9)bNoAlarms @RT(0) @T @F @DT @RT(4)BOOL @RT(0) @T @T @BASIC 0 @F
@F @F
@T
@BEG_Attrib
3 @RT(0) @RT(23)TRUE: no alarms are set @RT(0)
@END_Attrib
1 1 @F @F @F @F

@Var @RT(18)bCheckConditionsOk @RT(0) @T @F @DT @RT(4)BOOL @RT(0) @T @T @BASIC 0 @F
@F @F
@T
@BEG_Attrib
3 @RT(0) @RT(0) @RT(0)
@END_Attrib
1 3 @F @F @F @F

@Var @RT(23)bRelevantCheckCondition @RT(0) @T @F @DT @RT(4)BOOL @RT(0) @T @T @BASIC 0 @F
@F @F
@T
@BEG_Attrib
3 @RT(0) @RT(0) @RT(0)
@END_Attrib
1 0 @F @F @F @F

@Var @RT(16)iConditionsNotOk @RT(0) @T @F @DT @RT(4)DINT @RT(0) @T @T @BASIC 0 @F
@F @F
@T
@BEG_Attrib
3 @RT(0) @RT(39)number of not fulfilled checkconditions @RT(0)
@END_Attrib
1 3 @F @F @F @F

@END_Dcl

@END_Export

@BEG_Export

@BEG_Algo
@ALGORITHM @RT(27)aCheckStartConditionReached @STRUCTURED_TEXT
@RT(0) @RT(0) @RT(0) @F @F
@END_Algo

@BEG_Dcl
@RT(16)DclTreeContainer
7
@Var @RT(9)iInstance @RT(0) @T @F @DT @RT(4)DINT @RT(0) @T @T @BASIC 0 @F
@F @F
@T
@BEG_Attrib
3 @RT(0) @RT(26)instance of startcondition @RT(0)
@END_Attrib
1 1 @F @F @F @F

@Var @RT(8)bReached @RT(0) @T @F @DT @RT(4)BOOL @RT(0) @T @T @BASIC 0 @F
@F @F
@T
@BEG_Attrib
3 @RT(0) @RT(23)start condition reached @RT(0)
@END_Attrib
1 3 @F @F @F @F

@Var @RT(10)prActValue @RT(0) @T @T @REFTO 0 @T @DT @RT(4)REAL @RT(0) @T @T @BASIC 0 @F
@F @F
@T
@BEG_Attrib
3 @RT(0) @RT(49)reference to actual value of the related movement @RT(0)
@END_Attrib
1 0 @F @F @F @F

@Var @RT(20)pbReferenceCondition @RT(0) @T @T @REFTO 0 @T @DT @RT(4)BOOL @RT(0) @T @T @BASIC 0 @F
@F @F
@T
@BEG_Attrib
3 @RT(0) @RT(0) @RT(0)
@END_Attrib
1 0 @F @F @F @F

@Var @RT(9)Direction @RT(0) @T @T @DERIVED 0 @T @T @DT @RT(15)tnMoveDirection @RT(0) @T @T @UNKNOWN 0 @F
@F @F
@T
@BEG_Attrib
3 @RT(0) @RT(24)max to min or min to max @RT(0)
@END_Attrib
1 0 @F @F @F @F

@Var @RT(15)RelatedMovement @RT(0) @T @T @DERIVED 0 @T @T @DT @RT(9)KODC_Step @RT(0) @T @T @UNKNOWN 0 @F
@F @F
@T
@BEG_Attrib
3 @RT(0) @RT(0) @RT(0)
@END_Attrib
1 0 @F @F @F @F

@Var @RT(19)PrevRelatedMovement @RT(0) @T @T @DERIVED 0 @T @T @DT @RT(9)KODC_Step @RT(0) @T @T @UNKNOWN 0 @F
@F @F
@T
@BEG_Attrib
3 @RT(0) @RT(32)data from last call of algorithm @RT(0)
@END_Attrib
1 0 @F @F @F @F

@END_Dcl

@END_Export

@BEG_Export

@BEG_Algo
@ALGORITHM @RT(26)aCheckConditionSupervision @STRUCTURED_TEXT
@RT(0) @RT(0) @RT(0) @F @F
@END_Algo

@BEG_Dcl
@RT(16)DclTreeContainer
4
@Var @RT(9)iInstance @RT(0) @T @F @DT @RT(4)DINT @RT(0) @T @T @BASIC 0 @F
@F @F
@T
@BEG_Attrib
3 @RT(0) @RT(26)instance of startcondition @RT(0)
@END_Attrib
1 1 @F @F @F @F

@Var @RT(9)bContinue @RT(0) @T @F @DT @RT(4)BOOL @RT(0) @T @T @BASIC 0 @F
@F @F
@T
@BEG_Attrib
3 @RT(0) @RT(43)check condition must not be called any more @RT(0)
@END_Attrib
1 3 @F @F @F @F

@Var @RT(19)bTargetValueReached @RT(0) @T @F @DT @RT(4)BOOL @RT(0) @T @T @BASIC 0 @F
@F @F
@T
@BEG_Attrib
3 @RT(0) @RT(0) @RT(0)
@END_Attrib
1 0 @F @F @F @F

@Var @RT(12)fbLockUnlock @RT(0) @T @T @DERIVED 0 @T @T @DT @RT(12)FBLockUnlock @RT(0) @T @T @UNKNOWN 0 @F
@F @F
@T
@BEG_Attrib
3 @RT(0) @RT(0) @RT(0)
@END_Attrib
1 0 @F @F @F @F

@END_Dcl

@END_Export

@BEG_Export

@BEG_Algo
@ALGORITHM @RT(16)aCheckPosReached @STRUCTURED_TEXT
@RT(0) @RT(0) @RT(0) @F @F
@END_Algo

@BEG_Dcl
@RT(16)DclTreeContainer
11
@Var @RT(8)DeviceId @RT(0) @T @T @DERIVED 0 @T @T @DT @RT(10)tsDeviceId @RT(0) @T @T @UNKNOWN 0 @F
@F @F
@T
@BEG_Attrib
3 @RT(0) @RT(20)DeviceId of movement @RT(0)
@END_Attrib
1 1 @F @F @F @F

@Var @RT(6)MoveId @RT(0) @T @T @DERIVED 0 @T @T @DT @RT(10)tMoveIdent @RT(0) @T @T @UNKNOWN 0 @F
@F @F
@T
@BEG_Attrib
3 @RT(0) @RT(18)MoveId of movement @RT(0)
@END_Attrib
1 1 @F @F @F @F

@Var @RT(7)MoveDir @RT(0) @T @T @DERIVED 0 @T @T @DT @RT(10)tMoveIdent @RT(0) @T @T @UNKNOWN 0 @F
@F @F
@T
@BEG_Attrib
3 @RT(0) @RT(19)MoveDir of movement @RT(0)
@END_Attrib
1 1 @F @F @F @F

@Var @RT(7)iColumn @RT(0) @T @F @DT @RT(4)DINT @RT(0) @T @T @BASIC 0 @F
@F @F
@T
@BEG_Attrib
3 @RT(0) @RT(13)active column @RT(0)
@END_Attrib
1 1 @F @F @F @F

@Var @RT(4)iRow @RT(0) @T @F @DT @RT(4)DINT @RT(0) @T @T @BASIC 0 @F
@F @F
@T
@BEG_Attrib
3 @RT(0) @RT(10)active row @RT(0)
@END_Attrib
1 1 @F @F @F @F

@Var @RT(17)fbCheckPosReached @RT(0) @T @T @DERIVED 0 @T @T @DT @RT(17)FBCheckPosReached @RT(0) @T @T @UNKNOWN 0 @F
@F @F
@T
@BEG_Attrib
3 @RT(0) @RT(0) @RT(0)
@END_Attrib
1 0 @F @F @F @F

@Var @RT(17)fbMoveDescription @RT(0) @T @T @DERIVED 0 @T @T @DT @RT(17)FBMoveDescription @RT(0) @T @T @UNKNOWN 0 @F
@F @F
@T
@BEG_Attrib
3 @RT(0) @RT(0) @RT(0)
@END_Attrib
1 0 @F @F @F @F

@Var @RT(7)iMoveNr @RT(0) @T @F @DT @RT(4)DINT @RT(0) @T @T @BASIC 0 @F
@F @F
@T
@BEG_Attrib
3 @RT(0) @RT(0) @RT(0)
@END_Attrib
1 0 @F @F @F @F

@Var @RT(9)iInstance @RT(0) @T @F @DT @RT(4)DINT @RT(0) @T @T @BASIC 0 @F
@F @F
@T
@BEG_Attrib
3 @RT(0) @RT(0) @RT(0)
@END_Attrib
1 0 @F @F @F @F

@Var @RT(14)bPosNotReached @RT(0) @T @F @DT @RT(4)BOOL @RT(0) @T @T @BASIC 0 @F
@F @F
@T
@BEG_Attrib
3 @RT(0) @RT(0) @RT(0)
@END_Attrib
1 0 @F @F @F @F

@Var @RT(13)bPosReachedOk @RT(0) @T @F @DT @RT(4)BOOL @RT(0) @T @T @BASIC 0 @F
@F @F
@T
@BEG_Attrib
3 @RT(0) @RT(35)posReached ok -> cycle can continue @RT(0)
@END_Attrib
1 3 @F @F @F @F

@END_Dcl

@END_Export

@BEG_Export

@BEG_Algo
@ALGORITHM @RT(17)aCheckIfCondition @STRUCTURED_TEXT
@RT(0) @RT(0) @RT(0) @F @F
@END_Algo

@BEG_Dcl
@RT(16)DclTreeContainer
5
@Var @RT(9)iInstance @RT(0) @T @F @DT @RT(4)DINT @RT(0) @T @T @BASIC 0 @F
@F @F
@T
@BEG_Attrib
3 @RT(0) @RT(26)instance of IF - condition @RT(0)
@END_Attrib
1 1 @F @F @F @F

@Var @RT(12)bConditionOk @RT(0) @T @F @DT @RT(4)BOOL @RT(0) @T @T @BASIC 0 @F
@F @F
@T
@BEG_Attrib
3 @RT(0) @RT(26)TRUE: condition fullfilled @RT(0)
@END_Attrib
1 3 @F @F @F @F

@Var @RT(4)var1 @RT(0) @T @F @DT @RT(4)DINT @RT(0) @T @T @BASIC 0 @F
@F @F
@T
@BEG_Attrib
3 @RT(0) @RT(0) @RT(0)
@END_Attrib
1 0 @F @F @F @F

@Var @RT(4)var2 @RT(0) @T @F @DT @RT(4)DINT @RT(0) @T @T @BASIC 0 @F
@F @F
@T
@BEG_Attrib
3 @RT(0) @RT(0) @RT(0)
@END_Attrib
1 0 @F @F @F @F

@Var @RT(1)i @RT(0) @T @F @DT @RT(4)DINT @RT(0) @T @T @BASIC 0 @F
@F @F
@T
@BEG_Attrib
3 @RT(0) @RT(0) @RT(0)
@END_Attrib
1 0 @F @F @F @F

@END_Dcl

@END_Export

@BEG_Export

@BEG_Algo
@ALGORITHM @RT(19)aCheckLoopCondition @STRUCTURED_TEXT
@RT(0) @RT(0) @RT(0) @F @F
@END_Algo

@BEG_Dcl
@RT(16)DclTreeContainer
5
@Var @RT(9)iInstance @RT(0) @T @F @DT @RT(4)DINT @RT(0) @T @T @BASIC 0 @F
@F @F
@T
@BEG_Attrib
3 @RT(0) @RT(26)instance of IF - condition @RT(0)
@END_Attrib
1 1 @F @F @F @F

@Var @RT(12)bConditionOk @RT(0) @T @F @DT @RT(4)BOOL @RT(0) @T @T @BASIC 0 @F
@F @F
@T
@BEG_Attrib
3 @RT(0) @RT(26)TRUE: condition fullfilled @RT(0)
@END_Attrib
1 3 @F @F @F @F

@Var @RT(4)var1 @RT(0) @T @F @DT @RT(4)DINT @RT(0) @T @T @BASIC 0 @F
@F @F
@T
@BEG_Attrib
3 @RT(0) @RT(0) @RT(0)
@END_Attrib
1 0 @F @F @F @F

@Var @RT(4)var2 @RT(0) @T @F @DT @RT(4)DINT @RT(0) @T @T @BASIC 0 @F
@F @F
@T
@BEG_Attrib
3 @RT(0) @RT(0) @RT(0)
@END_Attrib
1 0 @F @F @F @F

@Var @RT(1)i @RT(0) @T @F @DT @RT(4)DINT @RT(0) @T @T @BASIC 0 @F
@F @F
@T
@BEG_Attrib
3 @RT(0) @RT(0) @RT(0)
@END_Attrib
1 0 @F @F @F @F

@END_Dcl

@END_Export

@BEG_Export

@BEG_Algo
@ALGORITHM @RT(10)aGoToEndIf @STRUCTURED_TEXT
@RT(0) @RT(0) @RT(0) @F @F
@END_Algo

@BEG_Dcl
@RT(16)DclTreeContainer
3
@Var @RT(7)iColumn @RT(0) @T @F @DT @RT(4)DINT @RT(0) @T @T @BASIC 0 @F
@F @F
@T
@BEG_Attrib
3 @RT(0) @RT(0) @RT(0)
@END_Attrib
1 1 @F @F @F @F

@Var @RT(8)iTmpLine @RT(0) @T @F @DT @RT(4)DINT @RT(0) @T @T @BASIC 0 @F
@F @F
@T
@BEG_Attrib
3 @RT(0) @RT(0) @RT(0)
@END_Attrib
1 4 @F @F @F @F

@Var @RT(6)iCount @RT(0) @T @F @DT @RT(3)INT @RT(0) @T @T @BASIC 0 @F
@F @F
@T
@BEG_Attrib
3 @RT(0) @RT(0) @RT(0)
@END_Attrib
1 0 @F @F @F @F

@END_Dcl

@END_Export

@BEG_Export

@BEG_Algo
@ALGORITHM @RT(12)aGoToEndLoop @STRUCTURED_TEXT
@RT(0) @RT(0) @RT(0) @F @F
@END_Algo

@BEG_Dcl
@RT(16)DclTreeContainer
3
@Var @RT(7)iColumn @RT(0) @T @F @DT @RT(4)DINT @RT(0) @T @T @BASIC 0 @F
@F @F
@T
@BEG_Attrib
3 @RT(0) @RT(0) @RT(0)
@END_Attrib
1 1 @F @F @F @F

@Var @RT(8)iTmpLine @RT(0) @T @F @DT @RT(4)DINT @RT(0) @T @T @BASIC 0 @F
@F @F
@T
@BEG_Attrib
3 @RT(0) @RT(0) @RT(0)
@END_Attrib
1 4 @F @F @F @F

@Var @RT(9)iInstance @RT(0) @T @F @DT @RT(4)DINT @RT(0) @T @T @BASIC 0 @F
@F @F
@T
@BEG_Attrib
3 @RT(0) @RT(13)loop instance @RT(0)
@END_Attrib
1 1 @F @F @F @F

@END_Dcl

@END_Export

@BEG_Export

@BEG_Algo
@ALGORITHM @RT(14)aGoToBeginLoop @STRUCTURED_TEXT
@RT(0) @RT(0) @RT(0) @F @F
@END_Algo

@BEG_Dcl
@RT(16)DclTreeContainer
3
@Var @RT(7)iColumn @RT(0) @T @F @DT @RT(4)DINT @RT(0) @T @T @BASIC 0 @F
@F @F
@T
@BEG_Attrib
3 @RT(0) @RT(0) @RT(0)
@END_Attrib
1 1 @F @F @F @F

@Var @RT(8)iTmpLine @RT(0) @T @F @DT @RT(4)DINT @RT(0) @T @T @BASIC 0 @F
@F @F
@T
@BEG_Attrib
3 @RT(0) @RT(0) @RT(0)
@END_Attrib
1 4 @F @F @F @F

@Var @RT(9)iInstance @RT(0) @T @F @DT @RT(4)DINT @RT(0) @T @T @BASIC 0 @F
@F @F
@T
@BEG_Attrib
3 @RT(0) @RT(13)loop instance @RT(0)
@END_Attrib
1 1 @F @F @F @F

@END_Dcl

@END_Export

@BEG_Export

@BEG_Algo
@ALGORITHM @RT(10)aInterpret @STRUCTURED_TEXT
@RT(0) @RT(0) @RT(0) @F @F
@END_Algo

@BEG_Dcl
@RT(16)DclTreeContainer
24
@Var @RT(7)fbStart @RT(0) @T @T @DERIVED 0 @T @T @DT @RT(7)FBStart @RT(0) @T @T @UNKNOWN 0 @F
@F @F
@T
@BEG_Attrib
3 @RT(0) @RT(0) @RT(0)
@END_Attrib
1 0 @F @F @F @F

@Var @RT(12)fbCheckReady @RT(0) @T @T @DERIVED 0 @T @T @DT @RT(12)FBCheckReady @RT(0) @T @T @UNKNOWN 0 @F
@F @F
@T
@BEG_Attrib
3 @RT(0) @RT(0) @RT(0)
@END_Attrib
1 0 @F @F @F @F

@Var @RT(17)fbCheckPosReached @RT(0) @T @T @DERIVED 0 @T @T @DT @RT(17)FBCheckPosReached @RT(0) @T @T @UNKNOWN 0 @F
@F @F
@T
@BEG_Attrib
3 @RT(0) @RT(0) @RT(0)
@END_Attrib
1 0 @F @F @F @F

@Var @RT(22)abODCCheckDependencies @RT(0) @T @T @DERIVED 0 @T @T @DT @RT(22)ABODCCheckDependencies @RT(0) @T @T @UNKNOWN 0 @F
@F @F
@T
@BEG_Attrib
3 @RT(0) @RT(0) @RT(0)
@END_Attrib
1 0 @F @F @F @F

@Var @RT(1)i @RT(0) @T @F @DT @RT(4)DINT @RT(0) @T @T @BASIC 0 @F
@F @F
@T
@BEG_Attrib
3 @RT(0) @RT(19)current step column @RT(0)
@END_Attrib
1 4 @F @F @F @F

@Var @RT(1)k @RT(0) @T @F @DT @RT(4)DINT @RT(0) @T @T @BASIC 0 @F
@F @F
@T
@BEG_Attrib
3 @RT(0) @RT(0) @RT(0)
@END_Attrib
1 4 @F @F @F @F

@Var @RT(4)iRow @RT(0) @T @F @DT @RT(4)DINT @RT(0) @T @T @BASIC 0 @F
@F @F
@T
@BEG_Attrib
3 @RT(0) @RT(12)current step @RT(0)
@END_Attrib
1 0 @F @F @F @F

@Var @RT(16)bConditionLinked @RT(0) @T @F @DT @RT(4)BOOL @RT(0) @T @T @BASIC 0 @F
@F @F
@T
@BEG_Attrib
3 @RT(0) @RT(0) @RT(0)
@END_Attrib
1 0 @F @F @F @F

@Var @RT(7)MoveDir @RT(0) @T @T @DERIVED 0 @T @T @DT @RT(10)tMoveIdent @RT(0) @T @T @UNKNOWN 0 @F
@F @F
@T
@BEG_Attrib
3 @RT(0) @RT(0) @RT(0)
@END_Attrib
1 0 @F @F @F @F

@Var @RT(6)MoveId @RT(0) @T @T @DERIVED 0 @T @T @DT @RT(10)tMoveIdent @RT(0) @T @T @UNKNOWN 0 @F
@F @F
@T
@BEG_Attrib
3 @RT(0) @RT(12)current step @RT(0)
@END_Attrib
1 0 @F @F @F @F

@Var @RT(8)DeviceId @RT(0) @T @T @DERIVED 0 @T @T @DT @RT(10)tsDeviceId @RT(0) @T @T @UNKNOWN 0 @F
@F @F
@T
@BEG_Attrib
3 @RT(0) @RT(12)current step @RT(0)
@END_Attrib
1 0 @F @F @F @F

@Var @RT(12)bIncreaseRow @RT(0) @T @F @DT @RT(4)BOOL @RT(0) @T @T @BASIC 0 @F
@F @F
@T
@BEG_Attrib
3 @RT(0) @RT(44)increase row pointer after handling movement @RT(0)
@END_Attrib
1 0 @F @F @F @F

@Var @RT(7)bJoinOK @RT(0) @T @F @DT @RT(4)BOOL @RT(0) @T @T @BASIC 0 @F
@F @F
@T
@BEG_Attrib
3 @RT(0) @RT(0) @RT(0)
@END_Attrib
1 0 @F @F @F @F

@Var @RT(12)iJoinsInLine @RT(0) @T @F @DT @RT(4)DINT @RT(0) @T @T @BASIC 0 @F
@F @F
@T
@BEG_Attrib
3 @RT(0) @RT(0) @RT(0)
@END_Attrib
1 0 @F @F @F @F

@Var @RT(24)evCheckLocklistEventData @RT(0) @T @T @DERIVED 0 @T @T @DT @RT(20)tevCheckLocklistData @RT(0) @T @T @UNKNOWN 0 @F
@F @F
@T
@BEG_Attrib
3 @RT(0) @RT(0) @RT(0)
@END_Attrib
1 0 @F @F @F @F

@Var @RT(8)MoveData @RT(0) @T @T @REFTO 0 @F @DERIVED 0 @T @T @DT @RT(10)tsMoveData @RT(0) @T @T @UNKNOWN 0 @F
@F @F
@T
@BEG_Attrib
3 @RT(0) @RT(0) @RT(0)
@END_Attrib
1 0 @F @F @F @F

@Var @RT(25)bNewSkipAlreadyPosReached @RT(0) @T @F @DT @RT(4)BOOL @RT(0) @T @T @BASIC 0 @F
@F @F
@T
@BEG_Attrib
3 @RT(0) @RT(0) @RT(0)
@END_Attrib
1 0 @F @F @F @F

@Var @RT(9)iInstance @RT(0) @T @F @DT @RT(4)DINT @RT(0) @T @T @BASIC 0 @F
@F @F
@T
@BEG_Attrib
3 @RT(0) @RT(0) @RT(0)
@END_Attrib
1 0 @F @F @F @F

@Var @RT(10)bGoToEndIf @RT(0) @T @F @DT @RT(4)BOOL @RT(0) @T @T @BASIC 0 @F
@F @F
@T
@BEG_Attrib
3 @RT(0) @RT(36)go to end_if movement in this column @RT(0)
@END_Attrib
1 0 @F @F @F @F

@Var @RT(12)bGoToEndLoop @RT(0) @T @F @DT @RT(4)BOOL @RT(0) @T @T @BASIC 0 @F
@F @F
@T
@BEG_Attrib
3 @RT(0) @RT(0) @RT(0)
@END_Attrib
1 0 @F @F @F @F

@Var @RT(14)bGoToBeginLoop @RT(0) @T @F @DT @RT(4)BOOL @RT(0) @T @T @BASIC 0 @F
@F @F
@T
@BEG_Attrib
3 @RT(0) @RT(0) @RT(0)
@END_Attrib
1 0 @F @F @F @F

@Var @RT(7)iTmpRow @RT(0) @T @F @DT @RT(4)DINT @RT(0) @T @T @BASIC 0 @F
@F @F
@T
@BEG_Attrib
3 @RT(0) @RT(0) @RT(0)
@END_Attrib
1 4 @F @F @F @F

@Var @RT(14)bMovementReady @RT(0) @T @F @DT @RT(4)BOOL @RT(0) @T @T @BASIC 0 @F
@F @F
@T
@BEG_Attrib
3 @RT(0) @RT(0) @RT(0)
@END_Attrib
1 0 @F @F @F @F

@Var @RT(28)bAllParallelOpenColumnsReady @RT(0) @T @F @DT @RT(4)BOOL @RT(0) @T @T @BASIC 0 @F
@F @F
@T
@BEG_Attrib
3 @RT(0) @RT(0) @RT(0)
@END_Attrib
1 0 @F @F @F @F

@END_Dcl

@END_Export

@BEG_Export

@BEG_Algo
@ALGORITHM @RT(10)aFindLabel @STRUCTURED_TEXT
@RT(0) @RT(0) @RT(0) @F @F
@END_Algo

@BEG_Dcl
@RT(16)DclTreeContainer
11
@Var @RT(8)DeviceId @RT(0) @T @T @DERIVED 0 @T @T @DT @RT(10)tsDeviceId @RT(0) @T @T @UNKNOWN 0 @F
@F @F
@T
@BEG_Attrib
3 @RT(0) @RT(38)DeviceId of the movement to search for @RT(0)
@END_Attrib
1 1 @F @F @F @F

@Var @RT(6)MoveId @RT(0) @T @T @DERIVED 0 @T @T @DT @RT(10)tMoveIdent @RT(0) @T @T @UNKNOWN 0 @F
@F @F
@T
@BEG_Attrib
3 @RT(0) @RT(36)MoveId of the movement to search for @RT(0)
@END_Attrib
1 1 @F @F @F @F

@Var @RT(7)MoveDir @RT(0) @T @T @DERIVED 0 @T @T @DT @RT(10)tMoveIdent @RT(0) @T @T @UNKNOWN 0 @F
@F @F
@T
@BEG_Attrib
3 @RT(0) @RT(37)MoveDir of the movement to search for @RT(0)
@END_Attrib
1 1 @F @F @F @F

@Var @RT(16)IntermediateCond @RT(0) @T @F @DT @RT(4)DINT @RT(0) @T @T @BASIC 0 @F
@F @F
@T
@BEG_Attrib
3 @RT(0) @RT(36)Intermediate condition to search for @RT(0)
@END_Attrib
1 1 @F @F @F @F

@Var @RT(19)bAllowNonMatchingId @RT(0) @T @F @DT @RT(4)BOOL @RT(0) @T @T @BASIC 0 @F
@F @F
@T
@BEG_Attrib
3 @RT(0) @RT(42)Also return a match if MoveId is different @RT(0)
@END_Attrib
1 1 @F @F @F @F

@Var @RT(14)SearchStartPos @RT(0) @T @T @DERIVED 0 @T @T @DT @RT(12)tsODCStepPos @RT(0) @T @T @UNKNOWN 0 @F
@F @F
@T
@BEG_Attrib
3 @RT(0) @RT(27)startposition for searching @RT(0)
@END_Attrib
1 1 @F @F @F @F

@Var @RT(7)StepPos @RT(0) @T @T @DERIVED 0 @T @T @DT @RT(12)tsODCStepPos @RT(0) @T @T @UNKNOWN 0 @F
@F @F
@T
@BEG_Attrib
3 @RT(0) @RT(49)Position in ODC array wher the movement was found @RT(0)
@END_Attrib
1 3 @F @F @F @F

@Var @RT(6)bFound @RT(0) @T @F @DT @RT(4)BOOL @RT(0) @T @T @BASIC 0 @F
@F @F
@T
@BEG_Attrib
3 @RT(0) @RT(28)TRUE if a movement was found @RT(0)
@END_Attrib
1 3 @F @F @F @F

@Var @RT(7)iTmpRow @RT(0) @T @F @DT @RT(4)DINT @RT(0) @T @T @BASIC 0 @F
@F @F
@T
@BEG_Attrib
3 @RT(0) @RT(0) @RT(0)
@END_Attrib
1 4 @F @F @F @F

@Var @RT(10)iTmpColumn @RT(0) @T @F @DT @RT(4)DINT @RT(0) @T @T @BASIC 0 @F
@F @F
@T
@BEG_Attrib
3 @RT(0) @RT(0) @RT(0)
@END_Attrib
1 4 @F @F @F @F

@Var @RT(13)iSearchColumn @RT(0) @T @F @DT @RT(4)DINT @RT(0) @T @T @BASIC 0 @F
@F @F
@T
@BEG_Attrib
3 @RT(0) @RT(0) @RT(0)
@END_Attrib
1 4 @F @F @F @F

@END_Dcl

@END_Export

@BEG_Export

@BEG_Algo
@ALGORITHM @RT(10)aSetInitOK @STRUCTURED_TEXT
@RT(0) @RT(0) @RT(0) @F @F
@END_Algo

@BEG_Dcl
@RT(16)DclTreeContainer
1
@Var @RT(11)DeviceIdAll @RT(0) @T @T @DERIVED 0 @T @T @DT @RT(10)tsDeviceId @RT(0) @T @T @UNKNOWN 0 @F
@F @F
@T
@BEG_Attrib
3 @RT(0) @RT(0) @RT(0)
@END_Attrib
1 0 @F @F @F @F

@END_Dcl

@END_Export

@BEG_Export

@BEG_Algo
@ALGORITHM @RT(7)aStatus @STRUCTURED_TEXT
@RT(0) @RT(0) @RT(0) @F @F
@END_Algo

@BEG_Dcl
@RT(16)DclTreeContainer
3
@Var @RT(7)bActive @RT(0) @T @F @DT @RT(4)BOOL @RT(0) @T @T @BASIC 0 @F
@F @F
@T
@BEG_Attrib
3 @RT(0) @RT(46)Interpreter is currently executing a ODC array @RT(0)
@END_Attrib
1 3 @F @F @F @F

@Var @RT(6)bError @RT(0) @T @F @DT @RT(4)BOOL @RT(0) @T @T @BASIC 0 @F
@F @F
@T
@BEG_Attrib
3 @RT(0) @RT(68)Interpreter is stopped, because a error happened during interpreting @RT(0)
@END_Attrib
1 3 @F @F @F @F

@Var @RT(9)bFinished @RT(0) @T @F @DT @RT(4)BOOL @RT(0) @T @T @BASIC 0 @F
@F @F
@T
@BEG_Attrib
3 @RT(0) @RT(63)Interpreter is stopped, because it reached the end of the array @RT(0)
@END_Attrib
1 3 @F @F @F @F

@END_Dcl

@END_Export

@BEG_Export

@BEG_Algo
@ALGORITHM @RT(18)aInterruptSequence @STRUCTURED_TEXT
@RT(0) @RT(0) @RT(0) @F @F
@END_Algo

@BEG_Dcl
@RT(16)DclTreeContainer
5
@Var @RT(16)StartedMovements @RT(0) @T @T @DERIVED 0 @T @T @DT @RT(28)tsStartedMoveDataODCExtended @RT(0) @T @T @UNKNOWN 0 @F
@F @F
@T
@BEG_Attrib
3 @RT(0) @RT(0) @RT(0)
@END_Attrib
1 0 @F @F @F @F

@Var @RT(6)fbStop @RT(0) @T @T @DERIVED 0 @T @T @DT @RT(6)FBStop @RT(0) @T @T @UNKNOWN 0 @F
@F @F
@T
@BEG_Attrib
3 @RT(0) @RT(0) @RT(0)
@END_Attrib
1 0 @F @F @F @F

@Var @RT(1)i @RT(0) @T @F @DT @RT(4)DINT @RT(0) @T @T @BASIC 0 @F
@F @F
@T
@BEG_Attrib
3 @RT(0) @RT(0) @RT(0)
@END_Attrib
1 4 @F @F @F @F

@Var @RT(7)iMoveNr @RT(0) @T @F @DT @RT(4)DINT @RT(0) @T @T @BASIC 0 @F
@F @F
@T
@BEG_Attrib
3 @RT(0) @RT(0) @RT(0)
@END_Attrib
1 0 @F @F @F @F

@Var @RT(15)fbGetMoveNumber @RT(0) @T @T @DERIVED 0 @T @T @DT @RT(15)FBGetMoveNumber @RT(0) @T @T @UNKNOWN 0 @F
@F @F
@T
@BEG_Attrib
3 @RT(0) @RT(0) @RT(0)
@END_Attrib
1 0 @F @F @F @F

@END_Dcl

@END_Export

@BEG_Export

@BEG_Algo
@ALGORITHM @RT(17)aContinueSequence @STRUCTURED_TEXT
@RT(0) @RT(0) @RT(0) @F @F
@END_Algo

@BEG_Dcl
@RT(16)DclTreeContainer
2
@Var @RT(1)i @RT(0) @T @F @DT @RT(4)DINT @RT(0) @T @T @BASIC 0 @F
@F @F
@T
@BEG_Attrib
3 @RT(0) @RT(0) @RT(0)
@END_Attrib
1 4 @F @F @F @F

@Var @RT(14)fbSetStepState @RT(0) @T @T @DERIVED 0 @T @T @DT @RT(14)FBSetStepState @RT(0) @T @T @UNKNOWN 0 @F
@F @F
@T
@BEG_Attrib
3 @RT(0) @RT(0) @RT(0)
@END_Attrib
1 0 @F @F @F @F

@END_Dcl

@END_Export

@BEG_Export

@BEG_Algo
@ALGORITHM @RT(15)aEnableNextStep @STRUCTURED_TEXT
@RT(0) @RT(0) @RT(0) @F @F
@END_Algo

@BEG_Dcl
@RT(16)DclTreeContainer
1
@Var @RT(1)i @RT(0) @T @F @DT @RT(4)DINT @RT(0) @T @T @BASIC 0 @F
@F @F
@T
@BEG_Attrib
3 @RT(0) @RT(0) @RT(0)
@END_Attrib
1 4 @F @F @F @F

@END_Dcl

@END_Export

@BEG_Export

@BEG_Algo
@ALGORITHM @RT(14)aResetStepMode @STRUCTURED_TEXT
@RT(0) @RT(0) @RT(0) @F @F
@END_Algo

@BEG_Dcl
@RT(16)DclTreeContainer
0
@END_Dcl

@END_Export

@BEG_Export

@BEG_Algo
@ALGORITHM @RT(12)aDecreaseRow @STRUCTURED_TEXT
@RT(0) @RT(0) @RT(0) @F @F
@END_Algo

@BEG_Dcl
@RT(16)DclTreeContainer
15
@Var @RT(18)bStartInActualLine @RT(0) @T @F @DT @RT(4)BOOL @RT(0) @T @T @BASIC 0 @F
@F @F
@T
@BEG_Attrib
3 @RT(0) @RT(61)TRUE: start in actual line; FALSE: start in (actual line - 1) @RT(0)
@END_Attrib
1 1 @F @F @F @F

@Var @RT(7)iColumn @RT(0) @T @F @DT @RT(4)DINT @RT(0) @T @T @BASIC 0 @F
@F @F
@T
@BEG_Attrib
3 @RT(0) @RT(0) @RT(0)
@END_Attrib
1 1 @F @F @F @F

@Var @RT(8)iTmpLine @RT(0) @T @F @DT @RT(4)DINT @RT(0) @T @T @BASIC 0 @F
@F @F
@T
@BEG_Attrib
3 @RT(0) @RT(0) @RT(0)
@END_Attrib
1 4 @F @F @F @F

@Var @RT(7)iEndRow @RT(0) @T @F @DT @RT(4)DINT @RT(0) @T @T @BASIC 0 @F
@F @F
@T
@BEG_Attrib
3 @RT(0) @RT(0) @RT(0)
@END_Attrib
1 1 @F @F @F @F

@Var @RT(7)iMoveId @RT(0) @T @T @DERIVED 0 @T @T @DT @RT(10)tMoveIdent @RT(0) @T @T @UNKNOWN 0 @F
@F @F
@T
@BEG_Attrib
3 @RT(0) @RT(0) @RT(0)
@END_Attrib
1 0 @F @F @F @F

@Var @RT(19)iNewActivatedColumn @RT(0) @T @F @DT @RT(4)DINT @RT(0) @T @T @BASIC 0 @F
@F @F
@T
@BEG_Attrib
3 @RT(0) @RT(0) @RT(0)
@END_Attrib
1 3 @F @F @F @F

@Var @RT(10)iTmpColumn @RT(0) @T @F @DT @RT(4)DINT @RT(0) @T @T @BASIC 0 @F
@F @F
@T
@BEG_Attrib
3 @RT(0) @RT(0) @RT(0)
@END_Attrib
1 4 @F @F @F @F

@Var @RT(14)fbSetStepState @RT(0) @T @T @DERIVED 0 @T @T @DT @RT(14)FBSetStepState @RT(0) @T @T @UNKNOWN 0 @F
@F @F
@T
@BEG_Attrib
3 @RT(0) @RT(0) @RT(0)
@END_Attrib
1 0 @F @F @F @F

@Var @RT(18)bParallelTreeReady @RT(0) @T @F @DT @RT(4)BOOL @RT(0) @T @T @BASIC 0 @F
@F @F
@T
@BEG_Attrib
3 @RT(0) @RT(0) @RT(0)
@END_Attrib
1 0 @F @F @F @F

@Var @RT(3)bOk @RT(0) @T @F @DT @RT(4)BOOL @RT(0) @T @T @BASIC 0 @F
@F @F
@T
@BEG_Attrib
3 @RT(0) @RT(0) @RT(0)
@END_Attrib
1 0 @F @F @F @F

@Var @RT(1)x @RT(0) @T @F @DT @RT(4)DINT @RT(0) @T @T @BASIC 0 @F
@F @F
@T
@BEG_Attrib
3 @RT(0) @RT(0) @RT(0)
@END_Attrib
1 4 @F @F @F @F

@Var @RT(19)bContinueDecreasing @RT(0) @T @F @DT @RT(4)BOOL @RT(0) @T @T @BASIC 0 @F
@F @F
@T
@BEG_Attrib
3 @RT(0) @RT(0) @RT(0)
@END_Attrib
1 0 @F @F @F @F

@Var @RT(9)iStartRow @RT(0) @T @F @DT @RT(4)DINT @RT(0) @T @T @BASIC 0 @F
@F @F
@T
@BEG_Attrib
3 @RT(0) @RT(0) @RT(0)
@END_Attrib
1 0 @F @F @F @F

@Var @RT(6)iCount @RT(0) @T @F @DT @RT(3)INT @RT(0) @T @T @BASIC 0 @F
@F @F
@T
@BEG_Attrib
3 @RT(0) @RT(0) @RT(0)
@END_Attrib
1 0 @F @F @F @F

@Var @RT(5)iLine @RT(0) @T @F @DT @RT(4)DINT @RT(0) @T @T @BASIC 0 @F
@F @F
@T
@BEG_Attrib
3 @RT(0) @RT(0) @RT(0)
@END_Attrib
1 4 @F @F @F @F

@END_Dcl

@END_Export

@BEG_Body
@TL(61)
(**************************************** WARNING ********************************************
 *** The KEBA Kemro K2 System including software is not intended for safety control tasks! ***
 ***                       For further information see Comment tab!                        ***
 *********************************************************************************************)

IF NOT bInitDone THEN
   dCycleTime := GET_TASK_INTERVAL();
   bInitDone := TRUE;
END_IF;

//check duration
//get timestamp for new movement and duration of last movement
IF sv_OperationMode >= nHalfAutomatic AND CHECK_REF(pMoveData^.pdCalculatedDuration^) THEN

   IF (pMoveData^.EditorData.MovementType <> nODCElementDuration) AND
      (pMoveData^.EditorData.MovementType <> nODCElementInstanceableDuration) THEN

      IF CHECK_REF (pMoveData^.pdStartDelaySet^) THEN
         dMovementDelay := pMoveData^.pdStartDelaySet^;
      ELSE
         dMovementDelay := t#0s;
      END_IF;

      fbRTC();
      dActTime := fbRTC.CDT;
      dDuration := dActTime - odcParallelInfo[iColumn].dStartTime - dMovementDelay;

      IF dDuration > t#1s THEN
         dDuration := dDuration + dCycleTime;
      END_IF;

      IF (dDuration > MULTIME(pMoveData^.pdCalculatedDuration^, 1.0 + sv_rMoveDurationTolerance/100.0)) OR
         (dDuration < MULTIME(pMoveData^.pdCalculatedDuration^, 1.0 - sv_rMoveDurationTolerance/100.0)) THEN

         //duration out of tolerance
         IF sv_TraceLevel.bODCInterpreter THEN
            rTmp1 := LINT_TO_REAL(TIME_TO_LINT(pMoveData^.pdCalculatedDuration^))/1000000.0;
            rTmp2 := LINT_TO_REAL(TIME_TO_LINT(dDuration))/1000000.0;
            dummy := Print('correcting duration of %d.%d %d/%d from %f to %f',
                           DeviceId.CompId, DeviceId.IndexId,
                           pMoveData^.MoveDir, pMoveData^.MoveId,
                           rTmp1, rTmp2);
         END_IF;

      ELSE
         //duration in tolerance
         sv_iDurationUpdateInTolerance := sv_iDurationUpdateInTolerance + 1;
      END_IF;

      //correct duration
      pMoveData^.pdCalculatedDuration^ := dDuration;

      IF pMoveData^.bInstanceable THEN
         //instanceable movement -> trigger editor update
         //for "normal" movement the update must be triggered in the according function unit
         fbUpdateProperties();
      END_IF;

   END_IF;
END_IF;

@END_Body

@@@BEG_Comment@@@
@TL(0)

@@@END_Comment@@@

@BEG_Body
@TL(19)
(**************************************** WARNING ********************************************
 *** The KEBA Kemro K2 System including software is not intended for safety control tasks! ***
 ***                       For further information see Comment tab!                        ***
 *********************************************************************************************)

//unlock all movements that were locked because of a check condition
FOR i := 1 TO cMaxCheckConditions DO
   IF mCheckCondHelpData[i].bMovementLocked THEN
      fbLockUnlock(DeviceId := mCheckCondHelpData[i].LockUnlockData.DeviceId,
                   MoveDir := mCheckCondHelpData[i].LockUnlockData.MoveDir,
                   MoveId := mCheckCondHelpData[i].LockUnlockData.MoveId,
                   Alarm := mCheckCondHelpData[i].LockUnlockData.Alarm,
                   Mode := nUnlock);

      mCheckCondHelpData[i].bMovementLocked := FALSE;
   END_IF;
END_FOR;

@END_Body

@@@BEG_Comment@@@
@TL(4)
Clear the internal ODC sequence array sv_ODCSequenceInt.
Needed when the sequence is reinitialized to make sure no remanents of a old sequence are left.

Each element in the safety array is set to cODCNoDependency
@@@END_Comment@@@

@BEG_Body
@TL(37)
(**************************************** WARNING ********************************************
 *** The KEBA Kemro K2 System including software is not intended for safety control tasks! ***
 ***                       For further information see Comment tab!                        ***
 *********************************************************************************************)

FOR i := 1 TO sv_iUsedColumns DO
   IF (bExcludeActiveColumns AND odcParallelInfo[i].bColumnActive) THEN
      ; //do not reset active columns
   ELSE
      odcParallelInfo[i].bColumnActive := FALSE;
      odcParallelInfo[i].bStartSent := FALSE;
      odcParallelInfo[i].bStartConditionWarnPrinted := FALSE;
      odcParallelInfo[i].bSkipAlreadyPosReached := FALSE;
      odcParallelInfo[i].bActivatedChecked := FALSE;
      odcParallelInfo[i].bPosReachedArrayLinked := FALSE;
      odcParallelInfo[i].bMovementReadyArrayLinked := FALSE;
      odcParallelInfo[i].bDisabled := FALSE;
      odcParallelInfo[i].iRow := 0;
   END_IF;
END_FOR;
